// TwinCAT 3 PLC project Sys1_Inbound
// ProgramVersion: 3.1.4026.26
// libraries:
//   Tc2_Standard, * (Beckhoff Automation GmbH)
//   Tc2_System, * (Beckhoff Automation GmbH)
// project tree:
//   DUTs/ Auto_Test_DB_DUT.TcDUT (not stored), Auto_Test_DUT.TcDUT (not stored), Barcode_Station_DUT.TcDUT (not stored), Charger_DUT.TcDUT (not stored), Gate_Station_DUT.TcDUT (not stored), Level_Keys_DUT.TcDUT
//   DUTs/Conveyors/ Buffer_Cnv_Control_DUT.TcDUT (not stored), Buffer_Cnv_Inputs_DUT.TcDUT (not stored), Buffer_Cnv_Settings_DUT.TcDUT (not stored), Cnv_Errors_DUT.TcDUT (not stored), Cnv_Inputs_DUT.TcDUT (not stored), Cnv_Instruction_DUT.TcDUT (not stored), Cnv_Level_Control_DUT.TcDUT (not stored), Cnv_Level_Inputs_DUT.TcDUT, Cnv_Level_Settings_DUT.TcDUT (not stored), Cnv_Motor_DUT.TcDUT (not stored), Cnv_VTD_Control_DUT.TcDUT (not stored), Cnv_VTD_Settings_DUT.TcDUT (not stored), ECnv_Control_DUT.TcDUT (not stored), ECnv_Settings_DUT.TcDUT
//   DUTs/Safety_Stops/ Sfts_Control_DUT.TcDUT, Sfts_Inputs_DUT.TcDUT, Sfts_Instruction_DUT.TcDUT (not stored), Sfts_Settings_DUT.TcDUT (not stored)
//   DUTs/System/ ID_Decoded_DUT.TcDUT (not stored), OrderTable_DUT.TcDUT (not stored), System_DUT.TcDUT (not stored), System_Settings_DUT.TcDUT (not stored), WMS_OPC_UA_DUT.TcDUT (not stored)
//   DUTs/VTD/ VTD_Control_DUT.TcDUT (not stored), VTD_Errors_DUT.TcDUT, VTD_Inputs_DUT.TcDUT (not stored), VTD_Instruction_DUT.TcDUT, VTD_Levels_DUT.TcDUT (not stored), VTD_Motor_DUT.TcDUT, VTD_Outputs_DUT.TcDUT (not stored), VTD_Settings_DUT.TcDUT (not stored), VTD_Shuttle_Interlock_DUT.TcDUT (not stored)
//   GVLs/ Bypass.TcGVL (not stored), CNV_HMI_IO.TcGVL (not stored), Control.TcGVL (not stored), Errors.TcGVL (not stored), Force.TcGVL (not stored), Settings.TcGVL (not stored), System_Control.TcGVL (not stored)
//   GVLs/HMI/ CNV_HMI.TcGVL (not stored)
//   GVLs/IO/ IO_Panel.TcGVL, IO_VFDs.TcGVL
//   / PlcTask.TcTTO (not stored)
//   POUs/Conveyors/ Buffer_Conveyor_FB.TcPOU
//   POUs/ MAIN.TcPOU (not stored), Stack_Lights_FB.TcPOU
//   POUs/System/ Conveyors_Transfer.TcPOU
//   POUs/System/Functions/ ID_Decode_F.TcPOU (not stored), Set_Bit_F.TcPOU
//   POUs/VTD/ Light_Bars_FB.TcPOU, VTD_FB.TcPOU
// real-time tasks:
//   TASK PlcTask: cycle T#10ms, priority 20, ADS port 350
//   TASK PlcTask1: cycle T#10ms, priority 21, ADS port 351
// I/O:
//   DEVICE VTD_1 (EtherCAT), AmsNetId 192.168.0.103.2.1
//     DI-01 (EPP1008-0022) [EPP1008-0022 8 Ch. Dig. Input 24V, 3ms, M12]
//     DI-02 (EPP1008-0022) [EPP1008-0022 8 Ch. Dig. Input 24V, 3ms, M12]
//     DI-03 (EPP1008-0022) [EPP1008-0022 8 Ch. Dig. Input 24V, 3ms, M12]
//     DI-04 (EPP1008-0022) [EPP1008-0022 8 Ch. Dig. Input 24V, 3ms, M12]
//     DI-05 (EPP1008-0022) [EPP1008-0022 8 Ch. Dig. Input 24V, 3ms, M12]
//     DI-06 (EPP1008-0022) [EPP1008-0022 8 Ch. Dig. Input 24V, 3ms, M12]
//     DI-07 (EPP1008-0022) [EPP1008-0022 8 Ch. Dig. Input 24V, 3ms, M12]
//     DI-08 (EPP1008-0022) [EPP1008-0022 8 Ch. Dig. Input 24V, 3ms, M12]
//     DI-09 (EPP1008-0022) [EPP1008-0022 8 Ch. Dig. Input 24V, 3ms, M12]
//     DI-10 (EPP1008-0022) [EPP1008-0022 8 Ch. Dig. Input 24V, 3ms, M12]
//     ENCODER (EPP5001-0002) [EPP5001-0002 1Ch. SSI Encoder]
//     DIO-01 (EPP2328-0002) [EPP2328-0002 4 CH. Dig. In, 3ms, 4 Ch. Dig. Out 24V, 2A, M12]
//     DIO-02 (EPP2328-0002) [EPP2328-0002 4 CH. Dig. In, 3ms, 4 Ch. Dig. Out 24V, 2A, M12]
//     DIO-03 (EPP2328-0002) [EPP2328-0002 4 CH. Dig. In, 3ms, 4 Ch. Dig. Out 24V, 2A, M12]
//     DIO-04 (EPP2328-0002) [EPP2328-0002 4 CH. Dig. In, 3ms, 4 Ch. Dig. Out 24V, 2A, M12]
//     DIO-05 (EPP2328-0002) [EPP2328-0002 4 CH. Dig. In, 3ms, 4 Ch. Dig. Out 24V, 2A, M12]
//     DIO-06 (EPP2328-0002) [EPP2328-0002 4 CH. Dig. In, 3ms, 4 Ch. Dig. Out 24V, 2A, M12]
//     DIO-07 (EPP2328-0002) [EPP2328-0002 4 CH. Dig. In, 3ms, 4 Ch. Dig. Out 24V, 2A, M12]
//     DI-11 (EPP1809-0022) [EPP1809-0022 16 Ch. Dig. Input 24V, 3ms, M8]
//     FDI-01 (EP1918-0002) [EP1918, 8Ch. Safety Input 24V, TwinSAFE]
//       modules: Module 1 (FSOE), Module 2 (FSLOGIC)
//     PLC_IOs (EK1200) [EK1200-5000 EtherCAT Power supply (2A E-Bus)]
//       DI-01 (EL1809) [EL1809 16Ch. Dig. Input 24V, 3ms]
//       DI-02 (EL1809) [EL1809 16Ch. Dig. Input 24V, 3ms]
//       DO-01 (EL2809) [EL2809 16Ch. Dig. Output 24V, 0.5A]
//       DO-02 (EL2809) [EL2809 16Ch. Dig. Output 24V, 0.5A]
//       F-PLC (EL6910) [EL6910, TwinSAFE PLC]
//       FDI-01 (EL1918) [EL1918, 8Ch. Safety Input 24V, TwinSAFE]
//         modules: Module 1 (FSOE), Module 2 (FSLOGIC)
//       FDO-01 (EL2912) [EL2912, 2Ch. Safety Output 24V, 2A, TwinSAFE]
//         modules: Module 1 (FSOE), Module 2 (FSOUT), Module 3 (DEVICEIO), Module 4 (FSLOGIC)
//       ETHERCAT-1 (EK1322) [EK1322 2-port EtherCAT P junction with feed-in]
//       ETHERCAT-2 (EK1322) [EK1322 2-port EtherCAT P junction with feed-in]
//       ETHERCAT-3 (EK1322) [EK1322 2-port EtherCAT P junction with feed-in]
//       PROFNET (EL6633) [EL6633 PROFINET IO Controller]
//       ETHERCAT-4 (EK1122) [EK1122 2 port EtherCAT junction]
//       POWER_SUPPLY (EL9410) [EL9410 E-Bus Power Supplier  (Diagnostics)]
//       END_TERMINAL (EL9011) [EL9011 End Terminal]
//   DEVICE MAIN (EtherCAT), AmsNetId 192.168.0.103.3.1
//     PLC_IOs (EK1200) [EK1200-5000 EtherCAT Power supply (2A E-Bus)]
//       DI-01 (EL1809) [EL1809 16Ch. Dig. Input 24V, 3ms]
//       DI-02 (EL1809) [EL1809 16Ch. Dig. Input 24V, 3ms]
//       DO-01 (EL2809) [EL2809 16Ch. Dig. Output 24V, 0.5A]
//       DO-02 (EL2809) [EL2809 16Ch. Dig. Output 24V, 0.5A]
//       F-PLC (EL6910) [EL6910, TwinSAFE PLC]
//       FDI-01 (EL1918) [EL1918, 8Ch. Safety Input 24V, TwinSAFE]
//         modules: Module 1 (FSOE), Module 2 (FSLOGIC)
//       FDI-02 (EL1918) [EL1918, 8Ch. Safety Input 24V, TwinSAFE]
//         modules: Module 1 (FSOE), Module 2 (FSLOGIC)
//       FDO-01 (EL2912) [EL2912, 2Ch. Safety Output 24V, 2A, TwinSAFE]
//         modules: Module 1 (FSOE), Module 2 (FSOUT), Module 3 (DEVICEIO), Module 4 (FSLOGIC)
//       FDO-02 (EL2912) [EL2912, 2Ch. Safety Output 24V, 2A, TwinSAFE]
//         modules: Module 1 (FSOE), Module 2 (FSOUT), Module 3 (DEVICEIO), Module 4 (FSLOGIC)
//       POWER_SUPPLY (EL9410) [EL9410 E-Bus Power Supplier  (Diagnostics)]
//       PROFNET (EL6633) [EL6633 PROFINET IO Controller]
//       ETHERCAT (EK1322) [EK1322 2-port EtherCAT P junction with feed-in]
//       END_TERMINAL (EL9011) [EL9011 End Terminal]

// ---- DUTs/Conveyors/Cnv_Level_Inputs_DUT.TcDUT
TYPE Cnv_Level_Inputs_DUT :
STRUCT
	Cnv1_Inputs:	Buffer_Cnv_Inputs_DUT;
	Cnv2_Inputs:	Buffer_Cnv_Inputs_DUT;
END_STRUCT
END_TYPE

// ---- DUTs/Conveyors/ECnv_Settings_DUT.TcDUT
TYPE ECnv_Settings_DUT :
STRUCT
	ID:	DINT;
	Barcode_ID:	UINT;
	Cnv_Level:	UINT;
	TC_Time:	UINT;
	Transfer_Time:	UINT;
	Pallet_Align_Time:	UINT;
	Slow_Speed:	UINT;
	Full_Speed:	UINT;
	Manual_Speed:	UINT;
END_STRUCT
END_TYPE

// ---- DUTs/Level_Keys_DUT.TcDUT
TYPE Level_Keys_DUT :
STRUCT
	Level:	ARRAY[1..6] OF BOOL;
END_STRUCT
END_TYPE

// ---- DUTs/Safety_Stops/Sfts_Control_DUT.TcDUT
TYPE Sfts_Control_DUT :
STRUCT
	Mode:  UINT;
	Error:  BOOL;
	Enabled:  Bool;
	Running:  Bool;
	LP_State:  USInt;
	Motor_Extend:  Bool;
	Motor_Retract:  Bool;
	SM_State:  UInt;
	Instruction:  Sfts_Instruction_DUT;
	Inputs:  Sfts_Inputs_DUT;
END_STRUCT
END_TYPE

// ---- DUTs/Safety_Stops/Sfts_Inputs_DUT.TcDUT
TYPE Sfts_Inputs_DUT :
STRUCT
	DP_Extended:  BOOL;
	DP_Retracted:  Bool;
END_STRUCT
END_TYPE

// ---- DUTs/VTD/VTD_Errors_DUT.TcDUT
TYPE VTD_Errors_DUT :
STRUCT
	Error_Word_1:	UINT;
	Error_Word_2:	UINT;
	Error_Word_3:	UINT;
	Error_Word_4:	UINT;
	Error_Word_5:	UINT;
END_STRUCT
END_TYPE

// ---- DUTs/VTD/VTD_Instruction_DUT.TcDUT
TYPE VTD_Instruction_DUT :
STRUCT
	Mode_Change:  UINT;
	Stop:  BOOL;
	Enable:  Bool;
	Execulte:  Bool;
	Reset:  Bool;
	Pallet_Type:  UInt;
	Task_ID:  UInt;
	Task_Metadata:  String;
	Move_To_Level:  UInt;
	Manual_Up:  Bool;
	Manual_Down:  Bool;
	Manual_LP_Retract:  Bool;
	Manual_LP_Extend:  Bool;
	Start_Teach:  BOOL;
END_STRUCT
END_TYPE

// ---- DUTs/VTD/VTD_Motor_DUT.TcDUT
TYPE VTD_Motor_DUT :
STRUCT
	Enable:  BOOL;
	Enabled:  BOOL;
	Ready:  Bool;
	Running:  Bool;
	Forward:  Bool;
	Reverse:  Bool;
	Brake_Opened:  Bool;
	Speed:  Int;
	Speed_Actual:  Int;
	Actual_Current:  Int;
	Actual_Torque:  UInt;
	Acc_Factor:  UInt;
	Config_Axis:  Word;
	Error:  Bool;
	Status:  Word;
	Communication_Error:  Word;
	Lockout:  BOOL;
END_STRUCT
END_TYPE

// ---- GVLs/IO/IO_Panel.TcGVL
{attribute 'qualified_only'}
VAR_GLOBAL
	C1112_VTD_CIRCUIT_BREAKER AT%I*:BOOL;
	

END_VAR

// ---- GVLs/IO/IO_VFDs.TcGVL
{attribute 'qualified_only'}
VAR_GLOBAL
	
END_VAR

// ---- POUs/Conveyors/Buffer_Conveyor_FB.TcPOU
FUNCTION_BLOCK Buffer_Conveyor_FB
VAR_INPUT
	Cnv_Settings:  Buffer_Cnv_Settings_DUT;
	VTD_Level:  UINT;
	Safety_OK:  Bool;
	CNV_In_Out:  Bool;
	CNV1_2_Selected:  UInt;
	Time_CheckPallet:  Time;
	Time_CheckNoPallet:  TIME;
END_VAR
VAR_OUTPUT
END_VAR
VAR_IN_OUT
	Cnv_Control:  Buffer_Cnv_Control_DUT;
END_VAR
VAR
	State:  UINT;
	Timer_Transfer:  TON;
	Watchdog:  TON;
	Transfer_Direction:  String;
	MainSetpoint:  Int;
	R_Automatic_Mode:  R_TRIG;
	R_Start_DB:  R_TRIG;
	R_Stop_DB:  R_TRIG;
	ID_Decoded:  ID_Decoded_DUT;
	ID_Decoded_From:  ID_Decoded_DUT;
	ID_Decoded_To:  ID_Decoded_DUT;
	T_Ramp:  TON;
	HMI_Reset:  Bool;
	T_CheckNoPallet:  TON;
	Time_SlowDown_Ramp:  Time;
	T_CheckPallet:  TON;
END_VAR
VAR_TEMP
	Execute_Old:  BOOL;
	Stop_Old:  BOOL;
	Forward:  Bool;
	Backward:  Bool;
	SftyPinUp:  Bool;
	SftyPinDown:  BOOL;
END_VAR

R_Start_DB(CLK := Cnv_Control.Instruction.Execute AND NOT Execute_Old);
R_Stop_DB(CLK := Cnv_Control.Instruction.Stop AND NOT Stop_Old);

Execute_Old := Cnv_Control.Instruction.Execute;
Stop_Old := Cnv_Control.Instruction.Stop;

Cnv_Control.Enabled := Cnv_Control.Instruction.Enable OR Cnv_Control.Mode = 3;

ID_Decode_F(ID := Cnv_Settings.ID,
            ID_Decoded := ID_Decoded);

ID_Decode_F(ID := Cnv_Control.Instruction.Transfer_From_ID,
              ID_Decoded := ID_Decoded_From);

ID_Decode_F(ID := Cnv_Control.Instruction.Transfer_To_ID,
              ID_Decoded := ID_Decoded_To);

//MODES
Cnv_Control.Mode := Cnv_Control.Instruction.Mode_Change;
IF (Cnv_Control.Mode = 1 OR Cnv_Control.Mode = 5) AND NOT Cnv_Control.Error THEN
    State := 500;
END_IF;

R_Automatic_Mode(CLK := Cnv_Control.Mode = 3);
IF R_Automatic_Mode.Q OR (NOT Cnv_Control.Enabled AND NOT Cnv_Control.Error) THEN
    State := 0;
END_IF;

(*
Mode select is done via the HMI. Might add external mode select switches.
        
        Mode select mask:
        0: Disabled
        1: Manual
        2: Semi-Auto
        3: Auto
        4: Teach - N/A for Cnv
        5: Maintenance
        
Device ID Format: XXYYZZ    
XX = Device type   
    40  VTD
    10  Cnv_Front_of_VTD
    11  Cnv_Rear_of_VTD
    12  Cnv_On_Extractor
    20  Safety_Stop_Front_of_VTD
    21  Safety_Stop_Rear_of_VTD
  
YY = Floor   
ZZ = VTD Connected to    
Example: 110203 Conveyor at the rear of VTD 3 on level 2    
*)

{REGION Sensor allocations}
    //PALLET DETECT
    Forward := Cnv_Control.Inputs.Forward_Sensor;
    Backward := Cnv_Control.Inputs.Backward_Sensor;
    
    //SAFETY PINS (IT DOESN'T EXIST IN ECONVEYORS)
    SftyPinUp := Cnv_Control.Safety_Stop_Cnrl.Inputs.DP_Extended;
    SftyPinDown := Cnv_Control.Safety_Stop_Cnrl.Inputs.DP_Retracted;
{END_REGION}

{REGION Cyclic Checks} 
    // Check Pallet
    T_CheckPallet(IN:=Forward AND Backward,
                   PT:=Time_CheckPallet);
    
    T_CheckNoPallet(IN:=Cnv_Control.Running AND NOT Forward AND NOT Backward,
                   PT:=Time_CheckNoPallet);
    
    //Conditions for Conveyor occupied
  IF T_CheckPallet.Q OR // Both sensors triggered after a timer
        (NOT Forward AND Backward AND NOT Cnv_Control.Running) OR //Forward sensor triggered and not running
        (Forward AND NOT Backward AND NOT Cnv_Control.Running) //Backward sensor triggered and not running
    THEN
        Cnv_Control.Cnv_Occupied := TRUE;//Conveyor occupied
    ELSIF T_CheckNoPallet.Q OR //Check pallet Timer
        (NOT Cnv_Control.Running AND NOT Forward AND NOT Backward) //No sensor detected and Conveyor not running
    THEN
        //No Pallet
        Cnv_Control.Cnv_Occupied := FALSE;
    END_IF;
    
    // Update the Cnv_Control opbject
    Cnv_Control.SM_State := State;
    Cnv_Control.Stopped := NOT Cnv_Control.Running;
    IF Cnv_Control.Instruction.Inbound_Ready OR Cnv_Control.Instruction.Outbound_Ready THEN
        Cnv_Control.Ready_For_Task := TRUE;
    ELSE
        Cnv_Control.Ready_For_Task := FALSE;
    END_IF;
    
    IF ID_Decoded.Device_Type = 10 THEN
        Settings.LCnv_Sys[ID_Decoded.VTD].Cnv_Level[ID_Decoded.Level].Cnv1.Cnv_Level := INT_TO_UINT(ID_Decoded.Level);
    ELSIF ID_Decoded.Device_Type = 11 THEN
        Settings.LCnv_Sys[ID_Decoded.VTD].Cnv_Level[ID_Decoded.Level].Cnv2.Cnv_Level := INT_TO_UINT(ID_Decoded.Level);
    END_IF;
{END_REGION}

{REGION Auto/Semi auto mode}
    CASE State OF
        0: //Initialization
            Cnv_Control.Instruction.Inbound_Ready := FALSE;
            Cnv_Control.Instruction.Outbound_Ready := FALSE;
            Cnv_Control.Instruction.Transfer_Complete := 0;
            Cnv_Control.Instruction.Transfer_in_Progress := FALSE;
            Cnv_Control.Running := FALSE;
            Cnv_Control.Motor.Forward := FALSE;
            Cnv_Control.Motor.Reverse := FALSE;
            Cnv_Control.Motor.Speed := 0;
            Timer_Transfer(IN := FALSE,
                            PT := T#0S);
            T_Ramp(IN := FALSE,
                    PT := t#0s);
            IF Cnv_Control.Enabled AND (Cnv_Control.Mode = 3 OR Cnv_Control.Mode = 2) AND Cnv_Control.Error = 0 THEN
                State := 10;
            END_IF;
            
        10: //Standby - Conveyor ready to receive instruction
            IF Cnv_Control.Ready_For_Task AND (R_Start_DB.Q OR Cnv_Control.Instruction.Start_Transfer)
            THEN //WCS NORMAL TRANSFER
                Cnv_Control.Instruction.Inbound_Ready := FALSE;
                Cnv_Control.Instruction.Outbound_Ready := FALSE;
                Cnv_Control.Done := FALSE;
                Cnv_Control.Running := TRUE;
                Cnv_Control.Instruction.Transfer_in_Progress := TRUE;
                Cnv_Control.Current_Task_ID := Cnv_Control.Instruction.Task_ID;
                State := 20;
            ELSIF Cnv_Control.Instruction.Start_Transfer AND ID_Decoded.Level = 10 AND VTD_Level <> Cnv_Settings.Cnv_Level THEN
                //Extractor not at the correct level
                Set_Bit_F(BIT_Number := 2,
                            Variavel := Cnv_Control.Cnv_Errors.Error_Word_3);
            END_IF;
            
            //----------------------- Pallet Movement -----------------------
        20: //Set the direction of transfer
            IF ID_Decoded.Device_Type = 10 AND ID_Decoded_From.Device_Type = 12 AND NOT Cnv_Control.Cnv_Occupied AND
                Control.ECnv_Sys[ID_Decoded.VTD].Cnv_Occupied THEN //Extractor to CNV 1
                Cnv_Control.Motor.Speed := Cnv_Settings.Full_Speed;
                Cnv_Control.Motor.Forward := TRUE;
                Transfer_Direction := 'Forward';
                State := 30;
            ELSIF ID_Decoded.Device_Type = 10 AND ID_Decoded_To.Device_Type = 11 AND Cnv_Control.Cnv_Occupied AND
                NOT Control.LCnv_Sys[ID_Decoded.VTD].Cnv_Level[ID_Decoded.Level].Cnv2.Cnv_Occupied THEN // CNV 1 to CNV 2
                IF Control.LCnv_Sys[ID_Decoded.VTD].Cnv_Level[ID_Decoded.Level].Cnv2.SM_State = 30 THEN //Wait CNV 2 Run
                    Cnv_Control.Motor.Speed := Cnv_Settings.Full_Speed;
                    Cnv_Control.Motor.Forward := TRUE;
                    Transfer_Direction := 'Forward';
                    State := 30;
                END_IF;
            ELSIF ID_Decoded.Device_Type = 11 AND ID_Decoded_To.Device_Type = 10 AND Cnv_Control.Cnv_Occupied AND
                NOT Control.LCnv_Sys[ID_Decoded.VTD].Cnv_Level[ID_Decoded.Level].Cnv1.Cnv_Occupied THEN //CNV 2 To Cnv 1
                IF Control.LCnv_Sys[ID_Decoded.VTD].Cnv_Level[ID_Decoded.Level].Cnv1.SM_State = 30 THEN //Wait CNV1 RUn
                    Cnv_Control.Motor.Speed := Cnv_Settings.Full_Speed;
                    Cnv_Control.Motor.Reverse := TRUE;
                    Transfer_Direction := 'Backward';
                    State := 30;
                END_IF;
            ELSIF ID_Decoded.Device_Type = 10 AND ID_Decoded_To.Device_Type = 12 AND Cnv_Control.Cnv_Occupied AND
                NOT Control.ECnv_Sys[ID_Decoded.VTD].Cnv_Occupied THEN //CNV 1 To extractor
                IF Control.ECnv_Sys[ID_Decoded.VTD].SM_State = 30 THEN //Wait CVTD RUn
                    Cnv_Control.Motor.Speed := Cnv_Settings.Full_Speed;
                    Cnv_Control.Motor.Reverse := TRUE;
                    Transfer_Direction := 'Backward';
                    State := 30;
                END_IF;
            ELSE //14:3 Cnv cannot transfer to that location
                Set_Bit_F(BIT_Number := 5,
                            Variavel := Cnv_Control.Cnv_Errors.Error_Word_2);
            END_IF;
            
        30: // Running
            IF R_Stop_DB.Q THEN
                Cnv_Control.Motor.Forward := FALSE;
                Cnv_Control.Motor.Reverse := FALSE;
                Cnv_Control.Motor.Speed := 0;
                State := 0;
            ELSE
                //Slowdown ramp
                T_Ramp(IN := TRUE,
                        PT := Time_SlowDown_Ramp);
                IF T_Ramp.ET > (Time_SlowDown_Ramp * 70) / 100 AND T_Ramp.ET < (Time_SlowDown_Ramp * 80) / 100 THEN
                    Cnv_Control.Motor.Speed := Cnv_Settings.Slow_Speed * 3;
                ELSIF T_Ramp.ET > (Time_SlowDown_Ramp * 80) / 100 AND T_Ramp.ET < (Time_SlowDown_Ramp * 90) / 100 THEN
                    Cnv_Control.Motor.Speed := Cnv_Settings.Slow_Speed * 2;
                ELSIF T_Ramp.ET >= Time_SlowDown_Ramp THEN
                    Cnv_Control.Motor.Speed := Cnv_Settings.Slow_Speed;
                END_IF;
            END_IF;
            
            //Check conditions to stop the motor
            IF (ID_Decoded.Device_Type = 10 AND ID_Decoded_From.Device_Type = 12) OR //ECONV To CNV 1 - 10(CNV1)
                (ID_Decoded.Device_Type = 11 AND ID_Decoded_From.Device_Type = 10) OR //CNV 1 To CNV 2 - 11(CNV2)
                (ID_Decoded.Device_Type = 10 AND ID_Decoded_From.Device_Type = 11) //CNV 2 To CNV 1 - 10(CNV1)
            THEN
                IF Cnv_Control.Cnv_Occupied THEN //Stop the motor if the conveyor is not occupied anymore
                    State := 35;
                END_IF;
            ELSIF (ID_Decoded.Device_Type = 10 AND ID_Decoded_To.Device_Type = 12) OR //CNV 1 To ECNV - 10(CNV1)
                (ID_Decoded.Device_Type = 10 AND ID_Decoded_To.Device_Type = 11) OR //CNV 1 To CNV 2 - 10(CNV1)
                (ID_Decoded.Device_Type = 11 AND ID_Decoded_To.Device_Type = 10) //CNV 2 To CNV 1 - 11(CNV2)
            THEN
                IF NOT Cnv_Control.Cnv_Occupied THEN //Stop the motor if the conveyor is occupied
                    State := 35;
                END_IF;
            END_IF;
            
            //Monitor the transfer progress
            Timer_Transfer(IN := TRUE,
                            PT := UINT_TO_TIME(Cnv_Settings.Transfer_Time) * 1000);
            //If the watchdog bites, kill the process
            IF Timer_Transfer.Q THEN //14:1 Transfer timed out
                Set_Bit_F(BIT_Number := 3,
                           Variavel := Cnv_Control.Cnv_Errors.Error_Word_2);
            END_IF;
            
        35: //Stop motor
                T_Ramp(IN := FALSE,
                        PT := T#0S);
                Cnv_Control.Motor.Forward := FALSE;
                Cnv_Control.Motor.Reverse := FALSE;
                Cnv_Control.Motor.Speed := 0;
                Cnv_Control.Done := TRUE;
                State := 0;
            
        //----------------------- Pallet Alignment -----------------------
        400: //Error state
            Cnv_Control.Instruction.Inbound_Ready := FALSE;
            Cnv_Control.Instruction.Outbound_Ready := FALSE;
            Cnv_Control.Running := FALSE;
            Cnv_Control.Motor.Speed := 0;
            Cnv_Control.Motor.Forward := FALSE;
            Cnv_Control.Motor.Reverse := FALSE;
            Cnv_Control.Instruction.Stop := FALSE;
            Cnv_Control.Instruction.Transfer_in_Progress := FALSE;
            Watchdog(IN := FALSE,
                      PT := T#0S);
            Timer_Transfer(IN := FALSE,
                            PT := T#0S);

            T_Ramp(IN := FALSE,
                    PT := t#0s);
            IF Cnv_Control.Instruction.Reset OR SYSTEM_CONTROL.Reset_All OR HMI_Reset THEN
                Cnv_Control.Warning := 0;
                Cnv_Control.Current_Task_ID := 0;
                Cnv_Control.Error := FALSE; //Reset the conveyor
                
                Cnv_Control.Cnv_Errors.Error_Word_1 := 0;
                Cnv_Control.Cnv_Errors.Error_Word_2 := 0;
                Cnv_Control.Cnv_Errors.Error_Word_3 := 0;
                Cnv_Control.Cnv_Errors.Error_Word_4 := 0;
                State := 0;
            END_IF;
            
        500:
            IF Cnv_Control.Enabled THEN
                IF Cnv_Control.Instruction.Foward OR
                    (ID_Decoded.Device_Type = 10 AND Cnv_Control.Instruction.Start_Transfer AND NOT CNV_In_Out AND CNV1_2_Selected = 1 (*RECEIVE = 0*)) OR
                    (ID_Decoded.Device_Type = 10 AND Cnv_Control.Instruction.Start_Transfer AND CNV_In_Out AND CNV1_2_Selected = 2 (*SEND = 1*)) OR
                    (ID_Decoded.Device_Type = 11 AND Cnv_Control.Instruction.Start_Transfer AND NOT CNV_In_Out AND NOT Forward (*RECEIVE = 0*))
                THEN
                    Cnv_Control.Motor.Speed := Cnv_Settings.Manual_Speed;
                    Cnv_Control.Motor.Forward := TRUE;
                    Cnv_Control.Running := TRUE;
                ELSIF Cnv_Control.Instruction.Backward OR
                    (ID_Decoded.Device_Type = 10 AND Cnv_Control.Instruction.Start_Transfer AND NOT CNV_In_Out AND CNV1_2_Selected = 2 (*RECEIVE = 0*)) OR
                    (ID_Decoded.Device_Type = 10 AND Cnv_Control.Instruction.Start_Transfer AND CNV_In_Out AND CNV1_2_Selected = 1 (*SEND = 1*)) OR
                    (ID_Decoded.Device_Type = 11 AND Cnv_Control.Instruction.Start_Transfer AND CNV_In_Out (*SEND = 1*))
                THEN
                    Cnv_Control.Motor.Speed := Cnv_Settings.Manual_Speed;
                    Cnv_Control.Motor.Reverse := TRUE;
                    Cnv_Control.Running := TRUE;
                ELSE
                    Cnv_Control.Motor.Speed := 0;
                    Cnv_Control.Motor.Forward := FALSE;
                    Cnv_Control.Motor.Reverse := FALSE;
                    Cnv_Control.Running := FALSE;
                END_IF;
            END_IF;
            IF Cnv_Control.Mode <> 1 AND Cnv_Control.Mode <> 5 THEN
                State := 0;
            END_IF;
    END_CASE;
{END_REGION}

{REGION Cyclic Error Checks}
    IF NOT Safety_OK THEN //11:1
        Set_Bit_F(BIT_Number := 0,
                    Variavel := Cnv_Control.Cnv_Errors.Error_Word_1);
    END_IF;
    
    IF Cnv_Control.Motor.Error THEN
        Set_Bit_F(BIT_Number:= 0,
                  Variavel := Cnv_Control.Cnv_Errors.Error_Word_4);
    END_IF;
    
    IF Cnv_Control.Instruction.Stop THEN //HMI STOP
        Set_Bit_F(BIT_Number := 1,
                    Variavel := Cnv_Control.Cnv_Errors.Error_Word_1);
    END_IF;
    
    IF Cnv_Control.Safety_Stop_Cnrl.Error THEN
        Set_Bit_F(BIT_Number := 1,
                    Variavel := Cnv_Control.Cnv_Errors.Error_Word_4);
    END_IF;
    
    IF ((ID_Decoded.VTD = 1 AND ERRORS.Errors_Profinet_1.8) OR
        (ID_Decoded.VTD = 2 AND Errors_Profinet_3.7)) AND Cnv_Control.Mode <> 1
    THEN //Profinet error
        Set_Bit_F(BIT_Number := 3,
                    Variavel := Cnv_Control.Cnv_Errors.Error_Word_3);
    END_IF;
    
    
    // go to error state
    IF Cnv_Control.Cnv_Errors.Error_Word_1 <> 0 OR
        Cnv_Control.Cnv_Errors.Error_Word_2 <> 0 OR
        Cnv_Control.Cnv_Errors.Error_Word_3 <> 0 OR
        Cnv_Control.Cnv_Errors.Error_Word_4 <> 0
    THEN
        Cnv_Control.Error := TRUE;
        State := 400;
    END_IF;
{END_REGION}

{REGION VFD}
    //Status
    Cnv_Control.Motor.Ready := (Cnv_Control.Inputs.VFD_Status.%X0 OR Cnv_Control.Inputs.VFD_Status.%X1) AND NOT Cnv_Control.Motor.Error;
    Cnv_Control.Motor.Error := Cnv_Control.Inputs.VFD_Status.%X3 OR Cnv_Control.Inputs.VFD_Status.%X7 OR NOT Cnv_Control.Inputs.VFD_Status.%X13;
    Cnv_Control.Motor.Enabled := Cnv_Control.Inputs.VFD_Status.%X2;
    Cnv_Control.Motor.Actual_Current := SCALE_X(MIN := 0,
                                                 VALUE := NORM_X(MIN := 0,
                                                                 VALUE := Cnv_Control.Inputs.VFD_ActualCurrent,
                                                                 MAX := 16384),
                                                 MAX := 1.98);
    
    
    //Actual Speed
    IF MainSetpoint > 0 THEN
        Cnv_Control.Motor.Speed_Actual := SCALE_X(MIN := 0,
                                                   VALUE := NORM_X(MIN := 0,
                                                                   VALUE := Cnv_Control.Inputs.VFD_Speed_Actual,
                                                                   MAX := 16384),
                                                   MAX := 130);
        
        Cnv_Control.Motor.Actual_Torque := SCALE_X(MIN := 0,
                                                    VALUE := NORM_X(MIN := 0,
                                                                    VALUE := Cnv_Control.Inputs.VFD_ActualTorque,
                                                                    MAX := 16384),
                                                    MAX := 100);
    ELSIF MainSetpoint < 0 THEN
        Cnv_Control.Motor.Speed_Actual := SCALE_X(MIN := 0,
                                                   VALUE := NORM_X(MIN := 0,
                                                                   VALUE := Cnv_Control.Inputs.VFD_Speed_Actual * -1,
                                                                   MAX := 16384),
                                                   MAX := 130);
        
        Cnv_Control.Motor.Actual_Torque := SCALE_X(MIN := 0,
                                                    VALUE := NORM_X(MIN := 0,
                                                                    VALUE := Cnv_Control.Inputs.VFD_ActualTorque * -1,
                                                                    MAX := 16384),
                                                    MAX := 100);
    ELSE
        Cnv_Control.Motor.Speed_Actual := 0;
        Cnv_Control.Motor.Actual_Torque := 0;
    END_IF;
    
    //MAIN SETPOINT
    IF Cnv_Control.Motor.Forward THEN
        MainSetpoint := (SCALE_X(MIN := 0,
                                  VALUE := NORM_X(MIN := 0,
                                                  VALUE := Cnv_Control.Motor.Speed (** 1.681*),
                                                  MAX := 130),
                                  MAX := 1865.0) * -1);
    ELSIF Cnv_Control.Motor.Reverse THEN
        MainSetpoint := SCALE_X(MIN := 0,
                                 VALUE := NORM_X(MIN := 0,
                                                 VALUE := Cnv_Control.Motor.Speed (** 1.681*),
                                                 MAX := 130),
                                 MAX := 1865.0);
    ELSE
        MainSetpoint := 0;
    END_IF;
    
    SinaSpeed(EnableAxis := Cnv_Control.Motor.Forward OR Cnv_Control.Motor.Reverse,
               AckError := Cnv_Control.Instruction.Reset OR "Reset_All" OR HMI_Reset,
               SpeedSp := MainSetpoint,
               RefSpeed := 1865.0,
               HWIDSTW := Cnv_Settings.G120_Hardware_ID,
               HWIDZSW := Cnv_Settings.G120_Hardware_ID);
{END_REGION}

HMI_Reset := "Screen_DB_1".Reset_All[1] OR "Screen_DB_1".Reset_All[2] OR "CNV_HMI"."Reset(1)"[1] OR "CNV_HMI"."Reset(1)"[2];
;

END_FUNCTION_BLOCK

// ---- POUs/System/Functions/Set_Bit_F.TcPOU
FUNCTION Set_Bit_F : BOOL
VAR_INPUT
	BIT_Number:  UINT;
END_VAR
VAR
END_VAR
VAR_IN_OUT
	Variavel: WORD;
END_VAR

// Set the bit
Variavel := Variavel OR SHL(WORD#1,BIT_Number);

END_FUNCTION

// ---- POUs/Stack_Lights_FB.TcPOU
FUNCTION_BLOCK Stack_Lights_FB
VAR_INPUT
	System_Auto:  BOOL;
	Fault:  BOOL;
END_VAR
VAR_OUTPUT
	Red:  BOOL;
	Green:  BOOL;
	Orange:  BOOL;
END_VAR
VAR
END_VAR

//Commands for Stack Light

IF Fault THEN  // Fault = Red
    Red := "Clock_0.5Hz";
    Green := FALSE;
    Orange := FALSE;
ELSIF System_Auto THEN  // (1)Manual = Yellow
    Orange := FALSE;
    Red := FALSE;
    Green := TRUE;
ELSIF NOT System_Auto THEN  // (2)Semi-Auto = Blue
    Green := FALSE;
    Orange := TRUE;
    Red := FALSE;
// ELSIF System_Auto = 3 THEN  // (3)Auto = Green
//     Green := FALSE;
//     Red := FALSE;
//     Yellow := TRUE;

ELSE
    Green := FALSE;
    Red := FALSE;
    Orange := FALSE;
END_IF;

END_FUNCTION_BLOCK

// ---- POUs/System/Conveyors_Transfer.TcPOU
FUNCTION Conveyors_Transfer : BOOL
VAR_INPUT
END_VAR
VAR
	i_Lev:  UINT;
	i_Sys:  UINT;
	Concat1:  String;
	Concat2:  String;
	ID:  DInt;
	StrLev:  String;
	StrSys:  String;
	Level:  UINT;
END_VAR

FOR i_Sys := 1 TO 2 DO
    StrSys := UINT_TO_STRING(i_Sys);
    // Remove "+"
    IF StrSys[1] = '+' THEN
        StrSys := RIGHT(StrSys, L := LEN(StrSys) - 1);
    END_IF;
    
    {region "ID OF THE VTD CONVEYOR"}
        FOR i_Lev := Settings.VTD_Sys[i_Sys].Lowest_Level TO Settings.VTD_Sys[i_Sys].Highest_Level DO
            IF (i_Sys >= 1) AND (i_Sys <= 2) THEN
                IF Control.VTD_Sys[i_Sys].Current_Level = i_Lev THEN
                    StrLev := UINT_TO_STRING(i_Lev);
                    
                    // Remove "+"
                    IF StrLev[1] = '+' THEN
                        StrLev := RIGHT(StrLev, L := LEN(StrLev) - 1);
                    END_IF;
                    
                    //Build ID
                    Concat1 := CONCAT('120', StrLev);
                    Concat2 := CONCAT(Concat1, '0');
                    ID := STRING_TO_DINT(CONCAT(Concat2, StrSys));
                    
                    Settings.ECnv_Sys[i_Sys].ID := ID;
                    Settings.ECnv_Sys[i_Sys].Cnv_Level := i_Lev;
                END_IF;
            END_IF;
        END_FOR;
    {endregion}
        
        {region "READY TO RECEIVE"}
            //EXTRACTOR CONVEYOR
            FOR i_Lev := 2 TO Settings.VTD_Sys[i_Sys].Highest_Level DO
                IF Control.VTD_Sys[i_Sys].Current_Level = i_Lev THEN
                    StrLev := UINT_TO_STRING(i_Lev);
                    
                    // Remove "+"
                    IF StrLev[1] = '+' THEN
                        StrLev := RIGHT(StrLev, L := LEN(StrLev) - 1);
                    END_IF;
                    
                    //Build ID
                    Concat1 := CONCAT('120', StrLev);
                    Concat2 := CONCAT(Concat1, '0');
                    ID := STRING_TO_DINT(CONCAT(Concat2, StrSys));
                END_IF;
                
                IF Settings.ECnv_Sys[i_Sys].ID = ID AND NOT Control.ECnv_Sys[i_Sys].Error AND NOT Control.ECnv_Sys[i_Sys].Running
                    AND NOT Control.ECnv_Sys[i_Sys].Cnv_Occupied AND NOT Control.ECnv_Sys[i_Sys].Instruction.Outbound_Ready AND
                    NOT Control.LCnv_Sys[i_Sys].Cnv_Level[i_Lev].Cnv1.Running AND
                    (Control.ECnv_Sys[i_Sys].Mode = 2 OR Control.ECnv_Sys[i_Sys].Mode = 3) THEN
                    Control.ECnv_Sys[i_Sys].Instruction.Inbound_Ready := TRUE;
                END_IF;
            END_FOR;
            
            //BUFFER CONVEYORS
            FOR i_Lev := 2 TO Settings.VTD_Sys[i_Sys].Highest_Level DO
                //CNV 1
                IF NOT Control.LCnv_Sys[i_Sys].Cnv_Level[i_Lev].Cnv1.Error AND
                    NOT Control.LCnv_Sys[i_Sys].Cnv_Level[i_Lev].Cnv1.Running AND
                    NOT Control.LCnv_Sys[i_Sys].Cnv_Level[i_Lev].Cnv1.Cnv_Occupied AND
                    NOT Control.LCnv_Sys[i_Sys].Cnv_Level[i_Lev].Cnv1.Instruction.Outbound_Ready AND
                    (Control.LCnv_Sys[i_Sys].Cnv_Level[i_Lev].Cnv1.Mode = 2 OR Control.LCnv_Sys[i_Sys].Cnv_Level[i_Lev].Cnv1.Mode = 3) AND
                    NOT Control.ECnv_Sys[i_Sys].Running AND NOT Control.LCnv_Sys[i_Sys].Cnv_Level[i_Lev].Cnv2.Running
                THEN
                    Control.LCnv_Sys[i_Sys].Cnv_Level[i_Lev].Cnv1.Instruction.Inbound_Ready := TRUE;
                END_IF;
                
                //CNV 2
                IF NOT Control.LCnv_Sys[i_Sys].Cnv_Level[i_Lev].Cnv2.Error AND
                    NOT Control.LCnv_Sys[i_Sys].Cnv_Level[i_Lev].Cnv2.Running AND
                    NOT Control.LCnv_Sys[i_Sys].Cnv_Level[i_Lev].Cnv2.Cnv_Occupied AND
                    NOT Control.LCnv_Sys[i_Sys].Cnv_Level[i_Lev].Cnv2.Instruction.Outbound_Ready AND
                    (Control.LCnv_Sys[i_Sys].Cnv_Level[i_Lev].Cnv2.Mode = 2 OR Control.LCnv_Sys[i_Sys].Cnv_Level[i_Lev].Cnv2.Mode = 3) THEN
                    Control.LCnv_Sys[i_Sys].Cnv_Level[i_Lev].Cnv2.Instruction.Inbound_Ready := TRUE;
                END_IF;
            END_FOR;
        {endregion}
        
        {region "READY TO SEND"}
            //EXTRACTOR CONVEYOR
            Level := Settings.ECnv_Sys[i_Sys].Cnv_Level;
            
            IF Settings.ECnv_Sys[i_Sys].Cnv_Level >= 2 AND
                Settings.ECnv_Sys[i_Sys].Cnv_Level <= Settings.VTD_Sys[i_Sys].Highest_Level AND //Leveled
                Control.ECnv_Sys[i_Sys].Cnv_Occupied AND //Econveyor occupied
                NOT Control.ECnv_Sys[i_Sys].Error AND //not error
                NOT Control.ECnv_Sys[i_Sys].Running AND //not RUNNING
                Control.LCnv_Sys[i_Sys].Cnv_Level[Level].Cnv1.Instruction.Inbound_Ready AND 
                (Control.LCnv_Sys[i_Sys].Cnv_Level[Level].Cnv1.Mode = 2 OR
                Control.LCnv_Sys[i_Sys].Cnv_Level[Level].Cnv1.Mode = 3)  AND //cnv1 semi or auto mode
                (Control.ECnv_Sys[i_Sys].Mode = 2 OR Control.ECnv_Sys[i_Sys].Mode = 3) THEN //Econveyor semi or auto mode 
                Control.ECnv_Sys[i_Sys].Instruction.Outbound_Ready := TRUE;
            END_IF;
            
            
            //BUFFER CONVEYORS
            FOR i_Lev := 2 TO Settings.VTD_Sys[i_Sys].Highest_Level DO
                //CNV 1
                IF ((Control.ECnv_Sys[i_Sys].Instruction.Inbound_Ready AND Control.VTD_Sys[i_Sys].Current_Level = i_Lev) OR
                    Control.LCnv_Sys[i_Sys].Cnv_Level[i_Lev].Cnv2.Instruction.Inbound_Ready) AND //Extractor or CNV 2, inbound ready
                    
                    NOT Control.LCnv_Sys[i_Sys].Cnv_Level[i_Lev].Cnv2.Instruction.Transfer_in_Progress AND //NOT CNV2 transfer in progress
                    Control.LCnv_Sys[i_Sys].Cnv_Level[i_Lev].Cnv1.Cnv_Occupied AND //Not occupied
                    NOT Control.LCnv_Sys[i_Sys].Cnv_Level[i_Lev].Cnv1.Error AND NOT Control.LCnv_Sys[i_Sys].Cnv_Level[i_Lev].Cnv1.Running AND //NOT error and NOT running
                    (Control.LCnv_Sys[i_Sys].Cnv_Level[i_Lev].Cnv1.Mode = 2 OR Control.LCnv_Sys[i_Sys].Cnv_Level[i_Lev].Cnv1.Mode = 3)//Semi auto or auto
                THEN 
                    Control.LCnv_Sys[i_Sys].Cnv_Level[i_Lev].Cnv1.Instruction.Outbound_Ready := TRUE;
                END_IF;
                
                //CNV 2
                IF Control.LCnv_Sys[i_Sys].Cnv_Level[i_Lev].Cnv1.Instruction.Inbound_Ready AND //CNV 1, inbound ready
                    NOT Control.LCnv_Sys[i_Sys].Cnv_Level[i_Lev].Cnv1.Instruction.Transfer_in_Progress AND //NOT CNV 1 transfer in progress
                    Control.LCnv_Sys[i_Sys].Cnv_Level[i_Lev].Cnv2.Cnv_Occupied AND //Not occupied
                    NOT Control.LCnv_Sys[i_Sys].Cnv_Level[i_Lev].Cnv2.Error AND NOT Control.LCnv_Sys[i_Sys].Cnv_Level[i_Lev].Cnv2.Running AND //NOT error and NOT running
                    (Control.LCnv_Sys[i_Sys].Cnv_Level[i_Lev].Cnv2.Mode = 2 OR Control.LCnv_Sys[i_Sys].Cnv_Level[i_Lev].Cnv2.Mode = 3)//Semi auto or auto
                THEN
                    Control.LCnv_Sys[i_Sys].Cnv_Level[i_Lev].Cnv2.Instruction.Outbound_Ready := TRUE;
                END_IF;
            END_FOR;
       {endregion}
    END_FOR;

END_FUNCTION

// ---- POUs/VTD/Light_Bars_FB.TcPOU
FUNCTION_BLOCK Light_Bars_FB
VAR_INPUT
	VTD_Mode:  UINT;
	VTD_Speed:  INT;
	Fault:  BOOL;
END_VAR
VAR_OUTPUT
	Animation_B1:  BYTE;
	Color_B1:  BYTE;
	Speed_B1:  Byte;
	Animation_B2:  Byte;
	Color_B2:  Byte;
	Speed_B2:  BYTE;
END_VAR
VAR
END_VAR

//Commands for Light Bar

IF VTD_Mode = 0 AND NOT Fault THEN // (0)Disabled = No light  
    Animation_B1:= Animation_B2:= 0;
    
ELSIF VTD_Mode = 1 AND VTD_Speed = 0 AND  NOT Fault AND NOT "SinaSpeed_VTD_DB_1".EnableAxis THEN // (1)Manual= Yellow Stop
    Animation_B1 := Animation_B2 := 1;
    Color_B1 := Color_B2 := 4;
    
ELSIF VTD_Mode = 1 AND VTD_Speed > 0 AND VTD_Speed <= 33 AND  NOT Fault AND "SinaSpeed_VTD_DB_1".EnableAxis THEN // (1)Manual= Yellow until 33%
    Animation_B1 := Animation_B2 := 2;
    Speed_B1 := Speed_B2 := 2;
    Color_B1 := Color_B2 := 4;
    
ELSIF VTD_Mode = 1 AND VTD_Speed > 33 AND VTD_Speed <= 100 AND  NOT Fault THEN // (1)Manual= Yellow until 66%
    Animation_B1 := Animation_B2 := 2;
    Speed_B1 := Speed_B2 := 0;
    Color_B1 := Color_B2 := 4;
    
// ELSIF VTD_Mode = 1 AND VTD_Speed > 66 AND VTD_Speed <= 100 AND  NOT Fault THEN // (1)Manual= Yellow until 100%
//     Animation_B1 := Animation_B2 := 2;
//     Speed_B1 := Speed_B2 := 1;
//     Color_B1 := Color_B2 := 4;
    
ELSIF VTD_Mode = 2 AND VTD_Speed = 0 AND  NOT Fault AND NOT "SinaSpeed_VTD_DB_1".EnableAxis THEN // (2)Semi-auto = Blue Stop
    Animation_B1 := Animation_B2 := 1;
    Color_B1 := Color_B2 := 9;
    Speed_B1 := Speed_B2 := 0;
    
ELSIF VTD_Mode = 2 AND VTD_Speed > 0 AND VTD_Speed <= 33 AND  NOT Fault AND "SinaSpeed_VTD_DB_1".EnableAxis THEN // (2)Semi-auto = Blue until 33%
    Animation_B1 := Animation_B2 := 2;
    Speed_B1 := Speed_B2 := 2;
    Color_B1 := Color_B2 := 9;
    
ELSIF VTD_Mode = 2 AND VTD_Speed > 33 AND VTD_Speed <= 100 AND  NOT Fault THEN // (2)Semi-auto = Blue until 66%
    Animation_B1 := Animation_B2 := 2;
    Speed_B1 := Speed_B2 := 0;
    Color_B1 := Color_B2 := 9;
    
// ELSIF VTD_Mode = 2 AND VTD_Speed > 66 AND VTD_Speed <= 100 AND  NOT Fault THEN // (2)Semi-auto = Blue until 100%
//     Animation_B1 := Animation_B2 := 2;
//     Speed_B1 := Speed_B2 := 1;
//     Color_B1 := Color_B2 := 9;
    
ELSIF VTD_Mode = 3 AND VTD_Speed = 0 AND  NOT Fault AND NOT "SinaSpeed_VTD_DB_1".EnableAxis THEN // (3)Auto = Green Stop
    Animation_B1 := Animation_B2 := 1;
    Color_B1 := Color_B2 := 0;
    
ELSIF VTD_Mode = 3 AND VTD_Speed > 0 AND VTD_Speed <= 33 AND  NOT Fault AND "SinaSpeed_VTD_DB_1".EnableAxis THEN // (3)Auto = Green until 33%
    Animation_B1 := Animation_B2 := 2;
    Speed_B1 := Speed_B2 := 2;
    Color_B1 := Color_B2 := 0;
    
ELSIF VTD_Mode = 3 AND VTD_Speed > 33 AND VTD_Speed <= 100 AND  NOT Fault THEN // (3)Auto = Green until 66%
    Animation_B1 := Animation_B2 := 2;
    Speed_B1 := Speed_B2 := 0;
    Color_B1 := Color_B2 := 0;
    
// ELSIF VTD_Mode = 3 AND VTD_Speed > 66 AND VTD_Speed <= 100 AND  NOT Fault THEN // (3)Auto = Green until 100%
//     Animation_B1 := Animation_B2 := 2;
//     Speed_B1 := Speed_B2 := 1;
//     Color_B1 := Color_B2 := 0;
    
ELSIF VTD_Mode = 4 AND VTD_Speed = 0 AND  NOT Fault THEN // (4)Tech = Orange Stop
    Animation_B1 := Animation_B2 := 1;
    Color_B1 := Color_B2 := 2;
    
ELSIF VTD_Mode = 4 AND VTD_Speed > 0 AND VTD_Speed <= 33 AND  NOT Fault THEN // (4)Tech = Orange until 33%
    Animation_B1 := Animation_B2 := 2;
    Speed_B1 := Speed_B2 := 2;
    Color_B1 := Color_B2 := 2;
    
ELSIF VTD_Mode = 4 AND VTD_Speed > 33 AND VTD_Speed <= 66 AND  NOT Fault THEN // (4)Tech = Orange until 66%
    Animation_B1 := Animation_B2 := 2;
    Speed_B1 := Speed_B2 := 0;
    Color_B1 := Color_B2 := 2;
    
ELSIF VTD_Mode = 4 AND VTD_Speed > 66 AND VTD_Speed <= 100 AND  NOT Fault THEN // (4)Tech = Orange until 100%
    Animation_B1 := Animation_B2 := 2;
    Speed_B1 := Speed_B2 := 1;
    Color_B1 := Color_B2 := 2;
    
ELSIF VTD_Mode = 5 AND VTD_Speed = 0 AND  NOT Fault THEN // (5)Maintenance = White Stop
    Animation_B1 := Animation_B2 := 1;
    Color_B1 := Color_B2 := 19;
    
ELSIF VTD_Mode = 5 AND VTD_Speed > 0 AND VTD_Speed <= 33 AND  NOT Fault THEN // (5)Maintenance = White until 33%
    Animation_B1 := Animation_B2 := 2;
    Speed_B1 := Speed_B2 := 2;
    Color_B1 := Color_B2 := 19;
    
ELSIF VTD_Mode = 5 AND VTD_Speed > 33 AND VTD_Speed <= 66 AND  NOT Fault THEN // (5)Maintenance = White until 66%
    Animation_B1 := Animation_B2 := 2;
    Speed_B1 := Speed_B2 := 0;
    Color_B1 := Color_B2 := 19;
    
ELSIF VTD_Mode = 5 AND VTD_Speed > 66 AND VTD_Speed <= 100 AND  NOT Fault THEN // (5)Maintenance = White until 100%
    Animation_B1 := Animation_B2 := 2;
    Speed_B1 := Speed_B2 := 1;
    Color_B1 := Color_B2 := 19;
    
ELSIF Fault THEN // Fault = Flash Red
    Animation_B1:= Animation_B2 := 2;
    Color_B1:=Color_B2 := 1;
END_IF;

END_FUNCTION_BLOCK

// ---- POUs/VTD/VTD_FB.TcPOU
FUNCTION_BLOCK VTD_FB
VAR_INPUT
	System_no:  UINT;
	Safety_OK:  BOOL;
	Cnv_Sensors:  Cnv_Inputs_DUT;
	VTD_Settings:  VTD_Settings_DUT;
	Bypass_DP:  BOOL;
// 	Bypass:  Safety_Bypass_RemotePanel;
END_VAR
VAR_OUTPUT
END_VAR
VAR_IN_OUT
	VTD_Control:  VTD_Control_DUT;
	LE_Bypass_HMI:  BOOL;
END_VAR
VAR
	State:  UINT;
	Last_State:  UINT;
	I_State:  UInt;
	LD_Timer_1:  TON;
	LD_Timer:  TON;
	DP_Timer:  TON;
	Watchdog:  TON;
	CS_TImer:  TON;
	Interlock_Timer:  TON;
	MainSetpoint:  Int;
	Position_Offset:  Real;
	ChangeToLow:  Array[1..4] of DInt;
	DestPosition:  Real;
	SetUpSpeed:  UInt;
	LevelBelowExtractor:  UInt;
	IEC_Timer_0_Instance:  TON;
	DestinationLevel:  UInt;
	CurrentlLevel:  UInt;
	VTD_ID_Decoded:  ID_Decoded_DUT;
	Cnv_ID_Decoded:  ARRAY[1..2] OF ID_Decoded_DUT;
	IEC_Timer_0_Instance_1:  TON;
	IEC_Timer_0_Instance_2:  TON;
	VTD_ControlInstructionTask_ID_Old:  Int;
	R_Execulte:  R_TRIG;
	R_AutomatcMode:  R_TRIG;
	T_Encoders_Difference:  TON;
	T_LE_Error:  TON;
	T_Setpoint_Delay:  TON;
	Distance_mm:  Real;
	TravelTime_s:  UInt;
	LE_Prev_mm:  Real;
	DeltaPos_mm:  Real;
	SampleTime_s:  Real;
	VTDSpeed_mm_s:  Real;
	T_Speed:  TON;
	Speed_mm_per_percent:  Real;
	Speed_mm_s:  Real;
	TravelTime_ms:  UInt;
	Watchdog_PT:  Time;
	Position_OLD:  Real;
	R_Position_OLD:  R_TRIG;
END_VAR

VAR_TEMP
	Level_Accuracy:  STRING;
	i:  UINT;
	Upper_limit:  Bool;
	Ultimate_SlowDown:  Bool;
	Ultimate_Creep:  Bool;
	Lower_Limit:  Bool;
	Level_Detect:  Bool;
	Level_Detect1:  Bool;
	Level_Detect2:  Bool;
	DP2_Extended:  Bool;
	DP2_Retracted:  Bool;
	DP1_Extended:  Bool;
	DP1_Retracted:  Bool;
	Chain_Slack_1:  Bool;
	Chain_Slack_2:  Bool;
	Chain_Slack_3:  Bool;
	Chain_Slack_4:  Bool;
	DP1_Retract:  Bool;
	DP1_Extend:  Bool;
	DP2_Retract:  Bool;
	DP2_Extend:  Bool;
	Cnvs1_NotExtended:  Bool;
	Cnvs2_NotExtended:  Bool;
	Stoppers_NotExtended:  Bool;
	MainSetpoint1:  Int;
	HMI_Reset:  BOOL;
END_VAR

//Execute
R_Execulte(CLK := VTD_Control.Instruction.Execulte);

IF VTD_Control.Mode = 3 THEN
    VTD_Control.Instruction.Enable := TRUE;
END_IF;

VTD_Control.Enabled := VTD_Control.Instruction.Enable;

VTD_Control.Mode := VTD_Control.Instruction.Mode_Change;

IF NOT VTD_Control.Enabled AND NOT VTD_Control.Error THEN
    State := 0;
END_IF;

//MANUAL MODE
IF (VTD_Control.Mode = 1 OR VTD_Control.Mode = 5) AND NOT VTD_Control.Error AND VTD_Control.Enabled THEN
    State := 500;
END_IF;

(*
TODO:

Mode select is done via the HMI. Might add external mode select switches.
        
        Mode select mask:
        0: Disabled
        1: Manual
        2: Semi-Auto
        3: Auto
        4: Teach
        5: Maintenance
        
Device ID Format: XXYYZZ    
XX = Device type   
    01   VTD
    10  Cnv_Front_of_VTD
    11  Cnv_Rear_of_VTD
    12  Cnv_On_Extractor
    20  Safety_Stop_Front_of_VTD
    21  Safety_Stop_Rear_of_VTD
YY = Floor   
ZZ = VTD Connected to 
*)

{region "Sensor allocations"}
    //Assign inputs to local vars
    Upper_limit := VTD_Control.Inputs.Upper_limit;
    Ultimate_SlowDown := VTD_Control.Inputs.Ultimate_SlowDown;
    Ultimate_Creep := VTD_Control.Inputs.Ultimate_Creep;
    Lower_Limit := VTD_Control.Inputs.Lower_Limit;
    Level_Detect1 := VTD_Control.Inputs.Level_Detect1;
    Level_Detect2 := VTD_Control.Inputs.Level_Detect2;
    DP1_Extended := VTD_Control.Inputs.DP1_Extended;
    DP1_Retracted := VTD_Control.Inputs.DP1_Retracted;
    DP2_Extended := VTD_Control.Inputs.DP2_Extended;
    DP2_Retracted := VTD_Control.Inputs.DP2_Retracted;
    Chain_Slack_1 := VTD_Control.Inputs.Chain_Slack_1;
    Chain_Slack_2 := VTD_Control.Inputs.Chain_Slack_2;
    Chain_Slack_3 := VTD_Control.Inputs.Chain_Slack_3;
    Chain_Slack_4 := VTD_Control.Inputs.Chain_Slack_4;
    VTD_Control.LinearEnc := VTD_Control.Inputs.LE_Position;
    VTD_Control.AE := VTD_Control.Inputs.AE_Position_1;
{endregion}

{region "Cyclic Checks"}
    // Check for Pallet
    IF Cnv_Sensors.Forward_Sensor OR Cnv_Sensors.Backward_Sensor THEN
        VTD_Control.Pallet_Loaded := 1;//'Unknown';
    ELSE
        //No Pallet
        VTD_Control.Pallet_Loaded := 0;//'None';
    END_IF;
    
    //Docking pins
        IF DP1_Extended AND DP2_Extended THEN
            VTD_Control.LP_State := 1; //'Extended'
        ELSIF DP1_Retracted AND DP2_Retracted THEN
            VTD_Control.LP_State := 2; //'Retracted'
        ELSE
            VTD_Control.LP_State := 0; //'Unknown'
        END_IF;
        
        VTD_Control.DP_Extended := VTD_Control.LP_State = 1;
    
    // Level detect
    Level_Detect := Level_Detect1 AND Level_Detect2;
    
    //VTD extractor is docked
    IF DP1_Extended AND DP2_Extended AND Level_Detect AND
        (VTD_Control.LinearEnc - VTD_Settings.Teach_Values.Levels_LE[LevelBelowExtractor]) <= VTD_Settings.Level_Detect_LE THEN
        VTD_Control.Docked := TRUE;
    ELSE
        VTD_Control.Docked := FALSE;
    END_IF;
    
    //Ultimate stop checks
    IF (VTD_Control.LinearEnc < VTD_Settings.Slowdown_Count_LE OR VTD_Control.LinearEnc > VTD_Settings.Teach_Values.Levels_LE[VTD_Settings.Highest_Level] - VTD_Settings.Slowdown_Count_LE) AND
        Ultimate_Creep AND Ultimate_SlowDown AND VTD_Control.Running THEN
        VTD_Control.Motor_Speed := VTD_Settings.Creep_Speed;
        VTD_Control.Warning := 3; // Overtravel creep zone reached
    ELSIF (VTD_Control.LinearEnc < VTD_Settings.Slowdown_Count_LE OR VTD_Control.LinearEnc > VTD_Settings.Teach_Values.Levels_LE[VTD_Settings.Highest_Level] - VTD_Settings.Slowdown_Count_LE) AND
        NOT Ultimate_Creep AND Ultimate_SlowDown AND VTD_Control.Running THEN
        VTD_Control.Motor_Speed := VTD_Settings.Slow_Speed; // Overtravel slow zone reached
    END_IF;
    
    //Update Variables
    IF VTD_Control.Current_Task_Type = 0 OR VTD_Control.Current_Task_Type = 1 THEN
        VTD_Control.SM_State := State;
    ELSIF VTD_Control.Current_Task_Type = 2 OR VTD_Control.Current_Task_Type = 3 THEN
        VTD_Control.SM_State := I_State;
    END_IF;
    
    FOR i := VTD_Settings.Lowest_Level TO VTD_Settings.Highest_Level DO
        IF NOT Control.LCnv_Sys[System_no].Cnv_Level[i].Cnv1.Safety_Stop_Cnrl.Inputs.DP_Extended THEN
            Cnvs1_NotExtended := true;
        END_IF;
        IF NOT Control.LCnv_Sys[System_no].Cnv_Level[i].Cnv2.Safety_Stop_Cnrl.Inputs.DP_Extended THEN
            Cnvs2_NotExtended := true;
        END_IF;
    END_FOR;
    
    //Confirm whish level is below the extractor
    FOR i := VTD_Settings.Lowest_Level TO VTD_Settings.Highest_Level DO
        IF VTD_Control.LinearEnc >= (VTD_Settings.Teach_Values.Levels_LE[i] - VTD_Settings.Level_Detect_LE) THEN
            LevelBelowExtractor := i;
        END_IF;
    END_FOR;
    
    Stoppers_NotExtended := Cnvs1_NotExtended (*AND Cnvs2_NotExtended*);
    
    //AE ERROR
    IF VTD_Control.Inputs.AE_Status_2.15 THEN
        VTD_Control.AE_Error := 1;
    ELSE
        VTD_Control.AE_Error := 0;
    END_IF;
    
    //Encoder Delta
    VTD_Control.Encoder_Delta := ABS(VTD_Control.AE - VTD_Control.LinearEnc);
    
    //CURRENT LEVEL
    FOR i := VTD_Settings.Lowest_Level TO VTD_Settings.Highest_Level DO
        IF ABS(VTD_Control.LinearEnc - VTD_Settings.Teach_Values.Levels_LE[i]) <= VTD_Settings.VTD_Level_Granularity AND Level_Detect THEN
            VTD_Control.Current_Level := i;
            EXIT;
        ELSE
            VTD_Control.Current_Level := 0;
        END_IF;
    END_FOR;
    
    //SPEED mm/S
    T_Speed(IN := TRUE,
             PT := T#100MS);
    
    IF T_Speed.Q THEN
        DeltaPos_mm := ABS(VTD_Control.LinearEnc - LE_Prev_mm);
        VTDSpeed_mm_s := DeltaPos_mm / SampleTime_s;
        LE_Prev_mm := VTD_Control.LinearEnc;
        T_Speed(IN := FALSE,
                 PT := T#0MS);
    END_IF;
{endregion}

{region "Auto/Semi-Auto Mode"}
    CASE State OF
        0: //Idle
            Last_State := State;
            VTD_Control.Motor_UP := FALSE;
            VTD_Control.Motor_Down := FALSE;
            VTD_Control.Motor.Speed := 0;
            DestinationLevel := CurrentlLevel := 0;
            VTD_Control.Stopped := TRUE;
            Watchdog(IN := FALSE,
                          PT := T#0S);
            IF VTD_Control.Mode = 3 OR VTD_Control.Mode = 2 THEN
                IF VTD_Control.Instruction.Enable AND NOT VTD_Control.Error THEN
                    State := 10;
                END_IF;
            END_IF;
            
        10: //Standby
            Last_State := State;
            IF VTD_Control.Enabled AND NOT VTD_Control.Running AND VTD_Control.Instruction.Move_To_Level >= VTD_Settings.Lowest_Level AND
                VTD_Control.Instruction.Move_To_Level <= VTD_Settings.Highest_Level AND VTD_Control.Pallet_Loaded <> 1 AND
                ((VTD_Control.Instruction.Task_ID > 0 OR VTD_Control.Instruction.Task_Metadata <> '' AND VTD_Control.Mode = 3 AND Control.VTD_Order_Table[System_no].Task_Type = 1) OR
                (VTD_Control.Mode = 2 (*AND R_Execulte.Q*)))
            THEN
                IF VTD_Control.Instruction.Move_To_Level = VTD_Control.Current_Level AND VTD_Control.Instruction.Move_To_Level <> 0 THEN
                    VTD_Control.Warning := 1; //VTD already at level requested
                    VTD_Control.Instruction.Move_To_Level := 0;
                    //Go straght to the travel complete feedabck 
                ELSIF ((VTD_Control.Shuttle_Loaded = 0 OR VTD_Control.Shuttle_Loaded = 1) AND System_no <= 3)
                    OR System_no > 3
                THEN //EVERYTHING OK
                    DestinationLevel := VTD_Control.Instruction.Move_To_Level;
                    CurrentlLevel := VTD_Control.Current_Level;
                    VTD_Control.Current_Task_ID := VTD_Control.Instruction.Task_ID;
                    VTD_Control.Running := TRUE;
                    State := 20;
                END_IF;
            END_IF;

        20: //Extend all safety stoppers that are not in the up position
            Last_State := State;
            VTD_Control.Done := FALSE;// To report to order table
            FOR i := VTD_Settings.Lowest_Level TO VTD_Settings.Highest_Level DO
                IF NOT Control.LCnv_Sys[System_no].Cnv_Level[i].Cnv1.Safety_Stop_Cnrl.Inputs.DP_Extended THEN
                    Control.LCnv_Sys[System_no].Cnv_Level[i].Cnv1.Safety_Stop_Cnrl.Instruction.Extend := TRUE;
                END_IF;
                IF NOT Control.LCnv_Sys[System_no].Cnv_Level[i].Cnv2.Safety_Stop_Cnrl.Inputs.DP_Extended THEN
                    Control.LCnv_Sys[System_no].Cnv_Level[i].Cnv2.Safety_Stop_Cnrl.Instruction.Extend := TRUE;
                END_IF;
            END_FOR;
            State := 25;
            
        25: //Check to ensure the Safety stoppers are in the up position.
            Last_State := State;
            FOR i := VTD_Settings.Lowest_Level TO VTD_Settings.Highest_Level DO
                IF Control.LCnv_Sys[System_no].Cnv_Level[i].Cnv1.Safety_Stop_Cnrl.Inputs.DP_Extended THEN
                    Control.LCnv_Sys[System_no].Cnv_Level[i].Cnv1.Safety_Stop_Cnrl.Instruction.Extend := FALSE;
                END_IF;
                IF Control.LCnv_Sys[System_no].Cnv_Level[i].Cnv2.Safety_Stop_Cnrl.Inputs.DP_Extended THEN
                    Control.LCnv_Sys[System_no].Cnv_Level[i].Cnv2.Safety_Stop_Cnrl.Instruction.Extend := FALSE;
                END_IF;
            END_FOR;
            
            IF Control.LCnv_Sys[System_no].Cnv_Level[2].Cnv1.Safety_Stop_Cnrl.Inputs.DP_Extended AND
                Control.LCnv_Sys[System_no].Cnv_Level[3].Cnv1.Safety_Stop_Cnrl.Inputs.DP_Extended AND
                Control.LCnv_Sys[System_no].Cnv_Level[4].Cnv1.Safety_Stop_Cnrl.Inputs.DP_Extended AND
                Control.LCnv_Sys[System_no].Cnv_Level[5].Cnv1.Safety_Stop_Cnrl.Inputs.DP_Extended AND
                Control.LCnv_Sys[System_no].Cnv_Level[6].Cnv1.Safety_Stop_Cnrl.Inputs.DP_Extended AND
                Control.LCnv_Sys[System_no].Cnv_Level[2].Cnv2.Safety_Stop_Cnrl.Inputs.DP_Extended AND
                Control.LCnv_Sys[System_no].Cnv_Level[3].Cnv2.Safety_Stop_Cnrl.Inputs.DP_Extended AND
                Control.LCnv_Sys[System_no].Cnv_Level[4].Cnv2.Safety_Stop_Cnrl.Inputs.DP_Extended AND
                Control.LCnv_Sys[System_no].Cnv_Level[5].Cnv2.Safety_Stop_Cnrl.Inputs.DP_Extended AND
                Control.LCnv_Sys[System_no].Cnv_Level[6].Cnv2.Safety_Stop_Cnrl.Inputs.DP_Extended
            THEN
                State := 30;
            END_IF;
            
        30: //Undock the VTD
            Last_State := State;
            IF LevelBelowExtractor >= VTD_Settings.Lowest_Level AND LevelBelowExtractor < VTD_Settings.Highest_Level THEN
                IF VTD_Control.Docked OR
                    (VTD_Control.LinearEnc < VTD_Settings.Teach_Values.Levels_LE[LevelBelowExtractor] + 50) OR
                    (VTD_Control.LinearEnc < VTD_Settings.Teach_Values.Levels_LE[LevelBelowExtractor + 1] AND
                    VTD_Control.LinearEnc > VTD_Settings.Teach_Values.Levels_LE[LevelBelowExtractor + 1] - 10) THEN
                    IF VTD_Control.LP_State = 1 THEN //extended
                        VTD_Control.Motor_Speed := VTD_Settings.Dock_speed;
                        VTD_Control.Motor_UP := TRUE;
                        Position_Offset := VTD_Control.LinearEnc + 40;
                        State := 35;
                    ELSIF VTD_Control.LP_State = 2 THEN //retracted
                        State := 45;
                    ELSE //24:4 Docking pins in an known state
                        Set_Bit_F(Bit_Number := 5,
                                    Bit_Value := 1,
                                    Variavel := VTD_Control.VTD_Errors.Error_Word_2);
                    END_IF;
                ELSE
                    Position_Offset := VTD_Control.LinearEnc - 5;
                    State := 35;
                END_IF;
            ELSIF LevelBelowExtractor = VTD_Settings.Highest_Level THEN
                IF VTD_Control.Docked OR
                    (VTD_Control.LinearEnc < VTD_Settings.Teach_Values.Levels_LE[LevelBelowExtractor] + 50) THEN
                    IF VTD_Control.LP_State = 1 THEN //extended
                        VTD_Control.Motor_Speed := VTD_Settings.Dock_speed;
                        VTD_Control.Motor_UP := TRUE;
                        Position_Offset := VTD_Control.LinearEnc + 40;
                        State := 35;
                    ELSIF VTD_Control.LP_State = 2 THEN //retracted
                        State := 45;
                    ELSE //24:4 Docking pins in an known state
                        Set_Bit_F(Bit_Number := 5,
                                    Variavel := VTD_Control.VTD_Errors.Error_Word_2);
                    END_IF;
                ELSE
                    Position_Offset := VTD_Control.LinearEnc - 5;
                    State := 35;
                END_IF;
            END_IF;
            
        35: //Stop motor
            Last_State := State;
            IF NOT Level_Detect AND VTD_Control.LinearEnc >= Position_Offset THEN
                VTD_Control.Motor_Speed := 0;
                VTD_Control.Motor_UP := FALSE;
                State := 36;
            END_IF;
            
        36: //Retract the docking pins
            Last_State := State;
                DP2_Retract := DP1_Retract := TRUE;
                DP_Timer(IN := TRUE,
                          PT := UINT_TO_TIME(VTD_Settings.Lockpins_Timeout_Retract));
                
                IF DP2_Retracted THEN
                    DP2_Retract := FALSE;
                END_IF;
                IF VTD_Control.Inputs.DP1_Retracted THEN
                    DP1_Retract := FALSE;
                END_IF;
                
                IF VTD_Control.LP_State = 2 THEN
                    State := 40;
                END_IF;
                
            40: //Check docking pins have been retracted
                Last_State := State;
            IF VTD_Control.LP_State = 2 THEN
                DP_Timer(IN := FALSE,
                          PT := T#0S);
                DP2_Retract := DP1_Retract := FALSE;
                State := 45;
            END_IF;
            
        45: //Start moving towards the level required
            Last_State := State;
            //Check load type and set extractor speed
            IF VTD_Control.Shuttle_Loaded = 0 AND VTD_Control.Pallet_Loaded = 0 THEN
                VTD_Control.Motor_Speed := VTD_Settings.Empty_Speed;
            ELSIF VTD_Control.Shuttle_Loaded = 1 AND VTD_Control.Pallet_Loaded = 0 THEN
                VTD_Control.Motor_Speed := VTD_Settings.Shuttle_Speed;
            ELSIF VTD_Control.Shuttle_Loaded = 0 AND (VTD_Control.Pallet_Loaded > 0) THEN
                VTD_Control.Motor_Speed := VTD_Settings.Pallet_Speed;
            ELSIF VTD_Control.Shuttle_Loaded = 1 AND (VTD_Control.Pallet_Loaded > 0) THEN
                VTD_Control.Motor_Speed := VTD_Settings.Loaded_Speed;
            END_IF;
            
            DestPosition := VTD_Settings.Teach_Values.Levels_LE[VTD_Control.Instruction.Move_To_Level];
            SetUpSpeed := VTD_Control.Motor_Speed;
            
            // === DINAMIC WATCHDOG ===
            Speed_mm_s := SetUpSpeed * Speed_mm_per_percent;
            Distance_mm := ABS(DestPosition - VTD_Control.LinearEnc);
            
            //VTD needs to move up
            IF VTD_Control.LinearEnc < DestPosition THEN
                VTD_Control.Motor_UP := TRUE;
                State := 50;
                //VTD needs to move down
            ELSIF VTD_Control.LinearEnc > DestPosition THEN
                VTD_Control.Motor_Down := TRUE;
                State := 65; //change to 65
            END_IF;
            
        50: //travel upwards to designated level
            Last_State := State;
            ChangeToLow[1] := ABS((VTD_Settings.Slowdown_Count_LE / 100) * 80); (* 80% *) //80  600mm
            ChangeToLow[2] := ABS((VTD_Settings.Slowdown_Count_LE / 100) * 60); (* 60% *) //60
            ChangeToLow[3] := ABS((VTD_Settings.Slowdown_Count_LE / 100) * 40); (* 40% *) //40
            ChangeToLow[4] := ABS((VTD_Settings.Slowdown_Count_LE / 100) * 20); (* 20% *) //20 60
            
            //switch to fast freq Low UP
            IF ABS(DestPosition - VTD_Control.LinearEnc) > VTD_Settings.Slowdown_Count_LE THEN
                VTD_Control.Motor_Speed := SetUpSpeed; //5
                //switch to low freq
            ELSIF ABS(DestPosition - VTD_Control.LinearEnc) <= VTD_Settings.Slowdown_Count_LE
                AND ABS(DestPosition - VTD_Control.LinearEnc) > ChangeToLow[1] THEN
                VTD_Control.Motor_Speed := VTD_Settings.Slow_Calib_Speed * 1.8; //5 * 1.8 = 9%
            ELSIF ABS(DestPosition - VTD_Control.LinearEnc) <= ChangeToLow[1]
                AND ABS(DestPosition - VTD_Control.LinearEnc) > ChangeToLow[2] THEN
                VTD_Control.Motor_Speed := VTD_Settings.Slow_Calib_Speed * 1.6; //5 * 1.6 = 8%
            ELSIF ABS(DestPosition - VTD_Control.LinearEnc) <= ChangeToLow[2]
                AND ABS(DestPosition - VTD_Control.LinearEnc) > ChangeToLow[3] THEN
                VTD_Control.Motor_Speed := VTD_Settings.Slow_Calib_Speed * 1.4; //5 * 1.4 = 7%
            ELSIF ABS(DestPosition - VTD_Control.LinearEnc) <= ChangeToLow[3]
                AND ABS(DestPosition - VTD_Control.LinearEnc) > ChangeToLow[4] THEN
                VTD_Control.Motor_Speed := VTD_Settings.Slow_Calib_Speed * 1.2; //5 * 1.2 = 6%
            ELSIF ABS(DestPosition - VTD_Control.LinearEnc) <= ChangeToLow[4] THEN
                VTD_Control.Motor_Speed := VTD_Settings.Slow_Calib_Speed; //5%
                State := 55;
            END_IF;
            
            // Timeout in ms
            IF Speed_mm_s > 0 THEN
                TravelTime_ms := REAL_TO_UINT((Distance_mm / Speed_mm_s) * 1500.0);  // 1.5x safety factor
                IF TravelTime_ms < 5000 THEN
                    TravelTime_ms := 5000; // mínimum 5s
                END_IF;
            ELSE
                TravelTime_ms := 30000; // fallback 30s 
            END_IF;
            
            Watchdog_PT := UINT_TO_TIME(TravelTime_ms);
            
            Watchdog.TON(IN := TRUE,
                          PT := Watchdog_PT);
            
            
        55: // Travel upwards using slow speed towards required floor
            Last_State := State;
            IF VTD_Control.LinearEnc > VTD_Settings.Teach_Values.Levels_LE[VTD_Control.Instruction.Move_To_Level] - VTD_Settings.Creep_Count_LE
            THEN
                VTD_Control.Motor_Speed := VTD_Settings.Creep_Speed; //3% - 60mm 
                State := 60;
            END_IF;
            
        60: // Travel past the level in order to extend the docking pins
            Last_State := State;
            IF VTD_Control.LinearEnc > VTD_Settings.Teach_Values.Levels_LE[VTD_Control.Instruction.Move_To_Level] + VTD_Settings.Creep_Count_LE
            THEN
                VTD_Control.Motor_Speed := 0;
                VTD_Control.Motor_UP := FALSE;
                VTD_Control.Motor_Down := FALSE;
                State := 80;
            END_IF;
            
        65: //travel Downwards to designated level   
            Last_State := State;
            ChangeToLow[1] := ABS((VTD_Settings.Slowdown_Count_LE / 100) * 80); (* 80% *) //80
            ChangeToLow[2] := ABS((VTD_Settings.Slowdown_Count_LE / 100) * 60); (* 60% *) //60
            ChangeToLow[3] := ABS((VTD_Settings.Slowdown_Count_LE / 100) * 40); (* 40% *) //40
            ChangeToLow[4] := ABS((VTD_Settings.Slowdown_Count_LE / 100) * 20); (* 20% *) //20
            //switch to fast freq Low UP
            IF ABS(DestPosition - VTD_Control.LinearEnc) > VTD_Settings.Slowdown_Count_LE THEN
                VTD_Control.Motor_Speed := SetUpSpeed;
                //switch to low freq
            ELSIF ABS(DestPosition - VTD_Control.LinearEnc) <= VTD_Settings.Slowdown_Count_LE
                AND ABS(DestPosition - VTD_Control.LinearEnc) > ChangeToLow[1] THEN
                VTD_Control.Motor_Speed := REAL_TO_UINT(VTD_Settings.Slow_Calib_Speed * 1.8);
            ELSIF ABS(DestPosition - VTD_Control.LinearEnc) <= ChangeToLow[1]
                AND ABS(DestPosition - VTD_Control.LinearEnc) > ChangeToLow[2] THEN
                VTD_Control.Motor_Speed := REAL_TO_UINT(VTD_Settings.Slow_Calib_Speed * 1.6);
            ELSIF ABS(DestPosition - VTD_Control.LinearEnc) <= ChangeToLow[2]
                AND ABS(DestPosition - VTD_Control.LinearEnc) > ChangeToLow[3] THEN
                VTD_Control.Motor_Speed := REAL_TO_UINT(VTD_Settings.Slow_Calib_Speed * 1.4);
            ELSIF ABS(DestPosition - VTD_Control.LinearEnc) <= ChangeToLow[3]
                AND ABS(DestPosition - VTD_Control.LinearEnc) > ChangeToLow[4] THEN
                VTD_Control.Motor_Speed := REAL_TO_UINT(VTD_Settings.Slow_Calib_Speed * 1.2);
            ELSIF ABS(DestPosition - VTD_Control.LinearEnc) <= ChangeToLow[4] THEN
                VTD_Control.Motor_Speed := VTD_Settings.Slow_Calib_Speed;
                State := 70;
            END_IF;
            
            // Timeout in ms
            IF Speed_mm_s > 0 THEN
                TravelTime_ms := REAL_TO_UINT((Distance_mm / Speed_mm_s) * 2000.0);  // 1.5x safety factor
                IF TravelTime_ms < 5000 THEN
                    TravelTime_ms := 5000; // mínimum 5s
                END_IF;
            ELSE
                TravelTime_ms := 30000; // fallback 30s 
            END_IF;
            
            Watchdog_PT := UINT_TO_TIME(TravelTime_ms);
            
            Watchdog(IN := TRUE,
                     PT := Watchdog_PT);
            
        70: // Travel downwards using slow speed towards required floor 
            Last_State := State;
            IF VTD_Control.LinearEnc < VTD_Settings.Teach_Values.Levels_LE[VTD_Control.Instruction.Move_To_Level] + VTD_Settings.Creep_Count_LE
            THEN
                VTD_Control.Motor_Speed := 0;
                VTD_Control.Motor_UP := FALSE;
                VTD_Control.Motor_Down := FALSE;
                State := 80;
            END_IF;
            
        80: //Extend Docking pins
            Last_State := State;
            IF VTD_Control.LP_State = 2 AND NOT Level_Detect THEN
                DP1_Extend := DP2_Extend := TRUE;
                DP_Timer(IN := TRUE,
                          PT := UINT_TO_TIME(VTD_Settings.Lockpins_Timeout_Extend));
            ELSIF VTD_Control.LP_State <> 1 AND NOT Level_Detect THEN
                DP1_Extend := DP2_Extend := TRUE;
            ELSIF VTD_Control.LP_State = 1 THEN
                State := 85;
            END_IF;
            
            
        85: // Wait for docking pins to extend
            Last_State := State;
            IF VTD_Control.LP_State = 1 AND NOT Level_Detect THEN
                DP_Timer(IN := FALSE,
                          PT := T#0S);
                DP1_Extend := DP2_Extend := FALSE;
                VTD_Control.Motor_Speed := VTD_Settings.Dock_speed;
                VTD_Control.Motor_Down := TRUE;
                State := 90;
            END_IF;
            
        90: // Dock the VTD
            Last_State := State;
            //Using the LE for comparation and Release tension in the VTD chain
            IF ABS(VTD_Control.LinearEnc - DestPosition) <= (VTD_Settings.Level_Detect_LE) AND NOT CS_TImer.Q THEN
                CS_TImer(IN := TRUE,
                          PT := UINT_TO_TIME(VTD_Settings.Chain_Slack_Timeout));
            END_IF;
            IF CS_TImer.Q THEN
                VTD_Control.Motor_Speed := 0;
                VTD_Control.Motor_Down := FALSE;
                CS_TImer(IN := FALSE,
                          PT := T#0S);
                State := 95;
            END_IF;
            
        95: // Dock the VTD
            Last_State := State;
            //Check the level detect sensors
            IF (Level_Detect1 AND NOT Level_Detect2) OR
                (NOT Level_Detect1 AND Level_Detect2) THEN
                LD_Timer(IN := TRUE,
                          PT := UINT_TO_TIME(VTD_Settings.Level_Detect_Timeout));
            ELSIF NOT Level_Detect1 AND NOT Level_Detect2 THEN
                LD_Timer_1(IN := TRUE,
                            PT := UINT_TO_TIME(VTD_Settings.Level_Detect_Timeout * 5));
            ELSE
                LD_Timer(IN := FALSE,
                          PT := T#0S);
                LD_Timer_1(IN := FALSE,
                            PT := T#0S);
            END_IF;
            
            IF Level_Detect THEN
                Watchdog(IN := FALSE,
                          PT := T#0S);
                State := 100;
            END_IF;
            
        100: //Wait for Movement completion ack  
            Last_State := State;
            //Reset timers
            VTD_Control.Instruction.Move_To_Level := 0;
            DP_Timer(IN := FALSE,
                      PT := T#0S);
            Watchdog(IN := FALSE,
                      PT := T#0S);
            LD_Timer(IN := FALSE,
                      PT := T#0S);
            CS_TImer(IN := FALSE,
                      PT := T#0S);
            LD_Timer_1(IN := FALSE,
                        PT := T#0S);
            
            VTD_Control.Motor_Speed := 0;
            VTD_Control.Current_Task_ID := 0;
            VTD_Control.Running := FALSE;
            State := 0;
            
        400: // Error state
            VTD_Control.Instruction.Move_To_Level := 0;
            VTD_Control.Done := FALSE;// To report to order table
            VTD_Control.Motor.Enable := FALSE;
            VTD_Control.Motor_UP := FALSE;
            VTD_Control.Motor_Down := FALSE;
            VTD_Control.Running := FALSE;
            VTD_Control.Stopped := TRUE;
            VTD_Control.Motor.Speed := 0;
            VTD_Control.Motor.Forward := FALSE;
            VTD_Control.Motor.Reverse := FALSE;
            DP1_Extend := DP2_Extend := FALSE;
            DP1_Retract := DP2_Retract := FALSE;
            FOR i := VTD_Settings.Lowest_Level TO VTD_Settings.Highest_Level DO
                Control.LCnv_Sys[System_no].Cnv_Level[i].Cnv1.Safety_Stop_Cnrl.Instruction.Extend := FALSE;
                Control.LCnv_Sys[System_no].Cnv_Level[i].Cnv2.Safety_Stop_Cnrl.Instruction.Extend := FALSE;
            END_FOR;
            //Reset timers
            DP_Timer(IN := FALSE,
                      PT := T#0S);
            Watchdog(IN := FALSE,
                      PT := T#0S);
            LD_Timer(IN := FALSE,
                      PT := T#0S);
            CS_TImer(IN := FALSE,
                      PT := T#0S);
            LD_Timer_1(IN := FALSE,
                        PT := T#0S);
            IF VTD_Control.Instruction.Reset OR Reset_All OR HMI_Reset THEN
                VTD_Control.Error := FALSE;
                VTD_Control.Warning := 0;
                VTD_Control.Stopped := FALSE;
                VTD_Control.Current_Task_Type := 0;
                VTD_Control.VTD_Errors.Error_Word_1 := 0;
                VTD_Control.VTD_Errors.Error_Word_2 := 0;
                VTD_Control.VTD_Errors.Error_Word_3 := 0;
                VTD_Control.VTD_Errors.Error_Word_4 := 0;
                VTD_Control.VTD_Errors.Error_Word_5 := 0;
                State := 0;
            END_IF;
            
        500: //MANUAL MODE
            IF VTD_Control.Error = 0 AND VTD_Control.Enabled THEN
                //VTD
                IF VTD_Control.Instruction.Manual_Up AND NOT Upper_limit THEN
                    VTD_Control.Motor_UP := TRUE;
                    VTD_Control.Stopped := FALSE;
                    VTD_Control.Running := TRUE;
                    IF NOT (Ultimate_SlowDown OR Ultimate_Creep) THEN
                        VTD_Control.Motor_Speed := VTD_Settings.Manual_Speed;
                    END_IF;
                ELSIF VTD_Control.Instruction.Manual_Down AND NOT Lower_Limit THEN
                    VTD_Control.Motor_Down := TRUE;
                    VTD_Control.Stopped := FALSE;
                    VTD_Control.Running := TRUE;
                    IF VTD_Control.LinearEnc <= VTD_Settings.Teach_Values.Levels_LE[LevelBelowExtractor] + 300 AND VTD_Control.LP_State = 1 THEN
                        VTD_Control.Motor_Speed := VTD_Settings.Creep_Speed;
                    ELSIF NOT (Ultimate_SlowDown OR Ultimate_Creep) THEN
                        VTD_Control.Motor_Speed := VTD_Settings.Manual_Speed;
                    END_IF;
                ELSE
                    VTD_Control.Motor_Speed := 0;
                    VTD_Control.Stopped := TRUE;
                    VTD_Control.Running := FALSE;
                    VTD_Control.Motor_Down := FALSE;
                    VTD_Control.Motor_UP := FALSE;
                END_IF;
                
                //DOCKING PINS 2 
                IF NOT VTD_Control.Running AND VTD_Control.Instruction.Manual_LP_Extend
                    AND NOT DP2_Extended THEN
                    DP2_Extend := TRUE;
                ELSIF NOT VTD_Control.Running AND VTD_Control.Instruction.Manual_LP_Retract
                    AND NOT DP2_Retracted THEN
                    DP2_Retract := TRUE;
                ELSE
                    DP2_Extend := FALSE;
                    DP2_Retract := FALSE;
                END_IF;
                
                //DOCKING PINS 1 
                IF NOT VTD_Control.Running AND VTD_Control.Instruction.Manual_LP_Extend
                    AND NOT DP1_Extended THEN
                    DP1_Extend := TRUE;
                ELSIF NOT VTD_Control.Running AND VTD_Control.Instruction.Manual_LP_Retract
                    AND NOT DP1_Retracted THEN
                    DP1_Retract := TRUE;
                ELSE
                    DP1_Extend := FALSE;
                    DP1_Retract := FALSE;
                END_IF;
                
                IF VTD_Control.Mode <> 1 AND VTD_Control.Mode <> 5 THEN
                    State := 0;
                END_IF;
                
                IF DP2_Extend OR DP1_Extend THEN
                    DP_Timer(IN := TRUE,
                              PT := UINT_TO_TIME(VTD_Settings.Lockpins_Timeout_Extend));
                ELSIF DP2_Retract OR DP1_Retract THEN
                    DP_Timer(IN := TRUE,
                              PT := UINT_TO_TIME(VTD_Settings.Lockpins_Timeout_Retract));
                ELSE
                    DP_Timer(IN := FALSE,
                              PT := T0S);
                END_IF;
            END_IF;
    END_CASE;
{endregion}

{region "Shuttle Interlock"}
    // VTD needs to be in Auto mode to perform a Shuttle interlock
    CASE I_State OF
        0:
            IF VTD_Control.Mode = 3 AND VTD_Control.Shuttle_Interlock.Interlock_Request AND VTD_Control.Shuttle_Interlock.Shuttle_Interlock_Task_ID > 0 THEN
                I_State := 10;
            END_IF;
            
        10: //Standby
            
            //Start by decoding all the IDs of the devices pertaining to the VTD in question on that level
            "ID_Decode_F"(ID := VTD_Settings.ID,
                          ID_Decoded := VTD_ID_Decoded);
            "ID_Decode_F"(ID := "Settings_DB".LCnv_Sys[System_no].Cnv_Level[VTD_Control.Current_Level].Cnv1.ID,
                          ID_Decoded := Cnv_ID_Decoded[1]);
            "ID_Decode_F"(ID := "Settings_DB".LCnv_Sys[System_no].Cnv_Level[VTD_Control.Current_Level].Cnv2.ID,
                          ID_Decoded := Cnv_ID_Decoded[2]);
            
            // Ensure the VTD is in a state that it can perform an interlock
            IF VTD_Control.Docked AND NOT VTD_Control.Running AND (VTD_Control.Shuttle_Loaded = 0 OR VTD_Control.Shuttle_Loaded = 1) AND VTD_Control.Error = 0 THEN
                // Check to make sure the VTD and Shuttle are not both loaded
                IF VTD_Control.Pallet_Loaded = 1 THEN
                    VTD_Control.Warning := 1; // Both the VTD and Shuttles are loaded, can't perform the interlock
                ELSE
                    //Check that shuttle is on the correct floor, that the start location given and the shuttle actual position matches and the destination is the correct extractor barcode
                    IF (*VTD_Control.Current_Level = "Shuttle_MQTT_DB".Shuttle_MQTT[VTD_Control.Shuttle_Interlock.Shuttle_ID].Message.Shuttle_Status.Floor
                            AND*)VTD_Control.Shuttle_Interlock.Shuttle_Start_Location = "Shuttle_MQTT_DB".Shuttle_MQTT[VTD_Control.Shuttle_Interlock.Shuttle_ID].Message.Shuttle_Status.Position_ID
                            (*AND "Shuttle_MQTT_DB".Shuttle_MQTT[VTD_Control.Shuttle_Interlock.Shuttle_ID].Message.Shuttle_Status.Destination_ID = "Settings_DB".ECnv_Settings.Barcode_ID*)THEN
                        
                        //Check in which Buffer conveyor the shuttle is located
                        IF "Settings_DB".LCnv_Sys[System_no].Cnv_Level[VTD_Control.Current_Level].Cnv1.Barcode_ID =
                            VTD_Control.Shuttle_Interlock.Shuttle_Start_Location THEN
                            VTD_Control.Running := TRUE;
                            I_State := 20;
                        ELSIF "Settings_DB".LCnv_Sys[System_no].Cnv_Level[VTD_Control.Current_Level].Cnv2.Barcode_ID =
                            VTD_Control.Shuttle_Interlock.Shuttle_Start_Location THEN
                            VTD_Control.Running := TRUE;
                            I_State := 25;
                        ELSIF "Settings_DB".ECnv_Sys[System_no].Barcode_ID =
                            VTD_Control.Shuttle_Interlock.Shuttle_Start_Location AND
                            Control_GVL.VTD_Order_Table[System_no].Destination_Location = "Settings_DB".LCnv_Sys[System_no].Cnv_Level[VTD_Control.Current_Level].Cnv1.Barcode_ID THEN
                            VTD_Control.Running := TRUE;
                            I_State := 20;
                        ELSIF "Settings_DB".ECnv_Sys[System_no].Barcode_ID =
                            VTD_Control.Shuttle_Interlock.Shuttle_Start_Location AND
                            Control_GVL.VTD_Order_Table[System_no].Destination_Location = "Settings_DB".LCnv_Sys[System_no].Cnv_Level[VTD_Control.Current_Level].Cnv2.Barcode_ID THEN
                            VTD_Control.Running := TRUE;
                            I_State := 25;
                        ELSE
                            VTD_Control.Warning := 2; // Shuttle interlock start location not buffer conveyor of VTD
                        END_IF;
                    ELSE
                        VTD_Control.Warning := 3; // Cant interlock as shuttle and VTD level mismatch
                    END_IF;
                END_IF;
            ELSE
                VTD_Control.Warning := 4; // VTD not ready for interlock 
            END_IF;
            
            
        20: //Drop safety stops
            IF Cnv_ID_Decoded[1].Level = VTD_Control.Current_Level THEN
                Control.LCnv_Sys[System_no].Cnv_Level[VTD_Control.Current_Level].Cnv1.Safety_Stop_Cnrl.Instruction.Retract := TRUE;
                I_State := 30;
            ELSE
                VTD_Control.Error := TRUE; //24:16 Cannot find the correct safety pins to drop.
                Set_Bit_F(Bit_Number := 1,
                            Bit_Value := 1,
                            Variavel := VTD_Control.VTD_Errors.Error_Word_3);
                // I_State := 400;
            END_IF;
            
        25: //Drop safety pins   
            IF Cnv_ID_Decoded[2].Level = VTD_Control.Current_Level THEN
                Control.LCnv_Sys[System_no].Cnv_Level[VTD_Control.Current_Level].Cnv2.Safety_Stop_Cnrl.Instruction.Retract := TRUE;
                I_State := 35;
            ELSE
                VTD_Control.Error := TRUE; //24:16 Cannot find the correct safety pins to drop.
                Set_Bit_F(Bit_Number := 1,
                            Bit_Value := 1,
                            Variavel := VTD_Control.VTD_Errors.Error_Word_3);
                // I_State := 400;
            END_IF;
            //////////////////////////////////////////////////////////////////////////////////////////////////////////////////////////////////////////////////////////////////    
        30: //Confirm safety stops are down at the correct location
            //Send ready to interlock
            IF Control.LCnv_Sys[System_no].Cnv_Level[VTD_Control.Current_Level].Cnv1.Safety_Stop_Cnrl.LP_State = 0 THEN //RETRACTED
                Control.LCnv_Sys[System_no].Cnv_Level[VTD_Control.Current_Level].Cnv1.Safety_Stop_Cnrl.Instruction.Retract := FALSE;
                VTD_Control.Shuttle_Interlock.Ready_To_Interlock := TRUE;
                I_State := 40;
            END_IF;
            
        35: //Confirm safety stops are down at the correct location
            //Send ready to interlock
            IF Control.LCnv_Sys[System_no].Cnv_Level[VTD_Control.Current_Level].Cnv2.Safety_Stop_Cnrl.LP_State = 0 THEN //RETRACTED
                Control.LCnv_Sys[System_no].Cnv_Level[VTD_Control.Current_Level].Cnv2.Safety_Stop_Cnrl.Instruction.Retract := FALSE;
                VTD_Control.Shuttle_Interlock.Ready_To_Interlock := TRUE;
                I_State := 45;
            END_IF;
            ////////////////////////////////////////////////////////////////////////////////////////////////////////////////////////////////////////////////////////////////////
        40: //Wait for shuttle to move in or out VTD
            IF Control_GVL.VTD_Order_Table[System_no].Destination_Location = "Settings_DB".ECnv_Sys[System_no].Barcode_ID THEN
                IF "Settings_DB".ECnv_Sys[System_no].Barcode_ID = "Shuttle_MQTT_DB".Shuttle_MQTT[VTD_Control.Shuttle_Interlock.Shuttle_ID].Message.Shuttle_Status.Position_ID
                    AND "Shuttle_MQTT_DB".Shuttle_MQTT[VTD_Control.Shuttle_Interlock.Shuttle_ID].Message.Shuttle_Status.Operational_State = 'IDLE' THEN
                    Control.LCnv_Sys[System_no].Cnv_Level[VTD_Control.Current_Level].Cnv1.Safety_Stop_Cnrl.Instruction.Extend := TRUE;
                    I_State := 50;
                END_IF;
            ELSIF Control.VTD_Order_Table[System_no].Destination_Location = "Settings_DB".LCnv_Sys[System_no].Cnv_Level[VTD_Control.Current_Level].Cnv1.Barcode_ID THEN
                IF "Settings_DB".LCnv_Sys[System_no].Cnv_Level[VTD_Control.Current_Level].Cnv1.Barcode_ID = "Shuttle_MQTT_DB".Shuttle_MQTT[VTD_Control.Shuttle_Interlock.Shuttle_ID].Message.Shuttle_Status.Position_ID
                    AND "Shuttle_MQTT_DB".Shuttle_MQTT[VTD_Control.Shuttle_Interlock.Shuttle_ID].Message.Shuttle_Status.Operational_State = 'IDLE' THEN
                    Control.LCnv_Sys[System_no].Cnv_Level[VTD_Control.Current_Level].Cnv1.Safety_Stop_Cnrl.Instruction.Extend := TRUE;
                    I_State := 50;
                END_IF;
            END_IF;
            
        45: //Wait for shuttle to move in or out VTD
            IF Control_GVL.VTD_Order_Table[System_no].Destination_Location = "Settings_DB".ECnv_Sys[System_no].Barcode_ID THEN
                IF "Settings_DB".ECnv_Sys[System_no].Barcode_ID = "Shuttle_MQTT_DB".Shuttle_MQTT[VTD_Control.Shuttle_Interlock.Shuttle_ID].Message.Shuttle_Status.Position_ID
                    AND "Shuttle_MQTT_DB".Shuttle_MQTT[VTD_Control.Shuttle_Interlock.Shuttle_ID].Message.Shuttle_Status.Operational_State = 'IDLE' THEN
                    Control.LCnv_Sys[System_no].Cnv_Level[VTD_Control.Current_Level].Cnv2.Safety_Stop_Cnrl.Instruction.Extend := TRUE;
                    I_State := 55;
                END_IF;
            ELSIF Control.VTD_Order_Table[System_no].Destination_Location = "Settings_DB".LCnv_Sys[System_no].Cnv_Level[VTD_Control.Current_Level].Cnv2.Barcode_ID THEN
                IF "Settings_DB".LCnv_Sys[System_no].Cnv_Level[VTD_Control.Current_Level].Cnv2.Barcode_ID = "Shuttle_MQTT_DB".Shuttle_MQTT[VTD_Control.Shuttle_Interlock.Shuttle_ID].Message.Shuttle_Status.Position_ID
                    AND "Shuttle_MQTT_DB".Shuttle_MQTT[VTD_Control.Shuttle_Interlock.Shuttle_ID].Message.Shuttle_Status.Operational_State = 'IDLE' THEN
                    Control.LCnv_Sys[System_no].Cnv_Level[VTD_Control.Current_Level].Cnv2.Safety_Stop_Cnrl.Instruction.Extend := TRUE;
                    I_State := 55;
                END_IF;
            END_IF;
            //////////////////////////////////////////////////////////////////////////////////////////////////////////////////////////////////////////////////////////////////////////  
        50: //Check own sensors for shuttle/pallet state
            IEC_Timer_0_Instance_1(IN := TRUE,
                                    PT := T5S);
            IF Control.LCnv_Sys[System_no].Cnv_Level[VTD_Control.Current_Level].Cnv1.Safety_Stop_Cnrl.LP_State = 1 //EXTENDED
                THEN
                Control.LCnv_Sys[System_no].Cnv_Level[VTD_Control.Current_Level].Cnv1.Safety_Stop_Cnrl.Instruction.Extend := FALSE;
                VTD_Control.Shuttle_Interlock.Interlock_Complete := TRUE;
                I_State := 60;
            ELSIF IEC_Timer_0_Instance_1.Q THEN
                VTD_Control.Error := TRUE; //24:17 Error occured during interlock final check
                Set_Bit_F(Bit_Number := 2,
                            Bit_Value := 1,
                            Variavel := VTD_Control.VTD_Errors.Error_Word_3);
                I_State := 400;
            END_IF;
            
        55: //Check own sensors for shuttle/pallet state
            IEC_Timer_0_Instance_1(IN := TRUE,
                                    PT := T5S);
            IF Control.LCnv_Sys[System_no].Cnv_Level[VTD_Control.Current_Level].Cnv2.Safety_Stop_Cnrl.LP_State = 1 //EXTENDED
                THEN
                Control.LCnv_Sys[System_no].Cnv_Level[VTD_Control.Current_Level].Cnv2.Safety_Stop_Cnrl.Instruction.Extend := FALSE;
                VTD_Control.Shuttle_Interlock.Interlock_Complete := TRUE;
                I_State := 60;
            ELSIF IEC_Timer_0_Instance_1.Q THEN
                VTD_Control.Error := TRUE; //24:17 Error occured during interlock final check
                Set_Bit_F(Bit_Number := 2,
                            Bit_Value := 1,
                            Variavel := VTD_Control.VTD_Errors.Error_Word_3);
                I_State := 400;
            END_IF;
            
        60://Clear Vars
            IEC_Timer_0_Instance_1(IN := FALSE,
                                    PT := T0s);
            IEC_Timer_0_Instance_2(IN := FALSE,
                                    PT := T0s);
            IF VTD_Control.Shuttle_Interlock.Interlock_Complete_Ack THEN
                VTD_Control.Shuttle_Interlock.Ready_To_Interlock := FALSE;
                VTD_Control.Shuttle_Interlock.Interlock_Complete := FALSE;
                VTD_Control.Running := FALSE;
                I_State := 0;
            END_IF;
            
        400://ERROR MODE
            IEC_Timer_0_Instance_1(IN := FALSE,
                                    PT := T#0S);
            IEC_Timer_0_Instance_2(IN := FALSE,
                                    PT := T#0S);
            Interlock_Timer(IN := FALSE,
                             PT := T#0S);
            VTD_Control.Running := FALSE;
            VTD_Control.Shuttle_Interlock.Interlock_Complete := FALSE;
            VTD_Control.Shuttle_Interlock.Ready_To_Interlock := FALSE;
            Control.LCnv_Sys[System_no].Cnv_Level[VTD_Control.Current_Level].Cnv1.Safety_Stop_Cnrl.Instruction.Extend := FALSE;
            Control.LCnv_Sys[System_no].Cnv_Level[VTD_Control.Current_Level].Cnv2.Safety_Stop_Cnrl.Instruction.Extend := FALSE;
            Control.LCnv_Sys[System_no].Cnv_Level[VTD_Control.Current_Level].Cnv1.Safety_Stop_Cnrl.Instruction.Retract := FALSE;
            Control.LCnv_Sys[System_no].Cnv_Level[VTD_Control.Current_Level].Cnv2.Safety_Stop_Cnrl.Instruction.Retract := FALSE;
            IF VTD_Control.Instruction.Reset THEN
                VTD_Control.VTD_Errors.Error_Word_3 := 0;
                I_State := 0;
            END_IF;
    END_CASE;
    Interlock_Timer(IN := I_State >= 40 AND I_State <= 50,
                     PT := UINT_TO_TIME("Settings_DB".System.Shuttle_Interlock_Timeout) * 1000);
    
{endregion}


// IF System_no <> 3 THEN
{region "Cyclic Error Checks"}
    IF NOT Safety_OK THEN //SAFETY
        Set_Bit_F(Bit_Number := 0,
                  Variavel := VTD_Control.VTD_Errors.Error_Word_1);
    END_IF;
    
    IF VTD_Control.Instruction.Stop THEN //HMI STOP
        Set_Bit_F(Bit_Number := 1,
                    Variavel := VTD_Control.VTD_Errors.Error_Word_1);
    END_IF;
    
    IF NOT VTD_Control.Inputs.Upper_Overtravel AND NOT Bypass.Upper_limit THEN //UPPER OVERTRAVEL
        Set_Bit_F(Bit_Number := 2,
                    Variavel := VTD_Control.VTD_Errors.Error_Word_1);
    END_IF;
    
    IF NOT VTD_Control.Inputs.Lower_Overtravel AND NOT Bypass.Lower_limit THEN //LOWER OVERTRAVEL
        Set_Bit_F(Bit_Number := 3,
                    Variavel := VTD_Control.VTD_Errors.Error_Word_1);
    END_IF;
    
    //CHAIN SLACK
    IF Chain_Slack_1 AND NOT Bypass.Chain_Slack_1 THEN
        Set_Bit_F(Bit_Number := 0,
                    Variavel := VTD_Control.VTD_Errors.Error_Word_5);
    END_IF;
    
    IF Chain_Slack_2 AND NOT Bypass.Chain_Slack_2 THEN
        Set_Bit_F(Bit_Number := 1,
                    Variavel := VTD_Control.VTD_Errors.Error_Word_5);
    END_IF;
    
    IF Chain_Slack_3 AND NOT Bypass.Chain_Slack_3 THEN
        Set_Bit_F(Bit_Number := 2,
                    Variavel := VTD_Control.VTD_Errors.Error_Word_5);
    END_IF;
    
    IF Chain_Slack_4 AND NOT Bypass.Chain_Slack_4 THEN
        Set_Bit_F(Bit_Number := 3,
                    Variavel := VTD_Control.VTD_Errors.Error_Word_5);
    END_IF;
    
    //VFD ERROR
    IF VTD_Control.Motor.Error THEN
        Set_Bit_F(Bit_Number := 7,
                    Variavel := VTD_Control.VTD_Errors.Error_Word_4);
    END_IF;
    
    //HIGH LIMITS
    IF VTD_Control.LinearEnc > VTD_Settings.VTD_Max_Heigh AND NOT LE_Bypass_HMI AND NOT "VTD_HMI".LE_Bypass[System_no] THEN //21:5
        Set_Bit_F(Bit_Number := 4,
                    Variavel := VTD_Control.VTD_Errors.Error_Word_1);
    END_IF;
    
    IF VTD_Control.LinearEnc < VTD_Settings.VTD_Min_Height AND NOT LE_Bypass_HMI AND NOT "VTD_HMI".LE_Bypass[System_no] THEN //21:5
        Set_Bit_F(Bit_Number := 5,
                    Variavel := VTD_Control.VTD_Errors.Error_Word_1);
    END_IF;
    
    //AUTOMATIC MODE NOT DOCKED
    R_AutomatcMode(CLK := VTD_Control.Mode = 3);
    IF NOT VTD_Control.Docked AND R_AutomatcMode.Q THEN //22:1
        Set_Bit_F(Bit_Number := 8,
                    Variavel := VTD_Control.VTD_Errors.Error_Word_1);
    END_IF;
    
    IF NOT Level_Detect AND R_AutomatcMode.Q THEN //22:2
        Set_Bit_F(Bit_Number := 9,
                    Variavel := VTD_Control.VTD_Errors.Error_Word_1);
    END_IF;
    
    //TRYING RETRACT WHILE DOCKED
    IF VTD_Control.Docked AND (DP1_Retract OR DP2_Retract) THEN //22:5
        Set_Bit_F(Bit_Number := 12,
                    Variavel := VTD_Control.VTD_Errors.Error_Word_1);
    END_IF;
    
    //LE ERROR
    T_LE_Error.TON(IN := VTD_Control.Inputs.LE_Status.%X0 OR VTD_Control.Inputs.LE_Status.%X1 OR
                    VTD_Control.LinearEnc < VTD_Settings.VTD_Min_Height OR
                    VTD_Control.LinearEnc > VTD_Settings.VTD_Max_Heigh,
                    PT := t500ms);
    IF NOT LE_Bypass_HMI AND NOT "VTD_HMI".LE_Bypass[System_no] AND T_LE_Error.Q THEN
        Set_Bit_F(Bit_Number := 4,
                    Variavel := VTD_Control.VTD_Errors.Error_Word_3);
        T_LE_Error.TON(IN := FALSE,
                        PT := T0s);
    END_IF;
    
    
    
    //ABSOLUTE ENCODER
    IF VTD_Control.AE_Error > 0 THEN
        Set_Bit_F(Bit_Number := 5,
                    Variavel := VTD_Control.VTD_Errors.Error_Word_3);
        VTD_Control.Outputs.AE_Control_Word_1.7 := VTD_Control.Instruction.Reset OR Reset_All OR HMI_Reset;
    ELSE
        VTD_Control.Outputs.AE_Control_Word_1.7 := FALSE;
    END_IF;
    
    IEC_Timer_0_Instance(IN := VTD_Control.LinearEnc <= (VTD_Settings.Teach_Values.Levels_LE[LevelBelowExtractor] + 1) AND VTD_Control.Instruction.Manual_Down,
                          PT := T#300MS);
    
    //Errors while running
    IF VTD_Control.Running THEN
        IF LevelBelowExtractor < 7 THEN
            IF NOT (VTD_Control.LP_State = 2) AND // NOT 'Retracted'
                (VTD_Control.LinearEnc > (VTD_Settings.Teach_Values.Levels_LE[LevelBelowExtractor] + VTD_Settings.Slowdown_Count_LE) AND
                VTD_Control.LinearEnc < (VTD_Settings.Teach_Values.Levels_LE[LevelBelowExtractor + 1] - VTD_Settings.Creep_Count_LE) AND
                VTD_Control.Instruction.Manual_Up)
                OR
                IEC_Timer_0_Instance.Q
            THEN //22:4
                IF NOT Bypass_LP THEN
                    IF System_no <> 5 THEN
                        Set_Bit_F(Bit_Number := 11,
                                    Variavel := VTD_Control.VTD_Errors.Error_Word_1);
                    END_IF;
                END_IF;
            END_IF;
        ELSIF LevelBelowExtractor = 8 THEN
            IF NOT (VTD_Control.LP_State = 2) AND // NOT 'Retracted'
                (VTD_Control.LinearEnc > (VTD_Settings.Teach_Values.Levels_LE[LevelBelowExtractor] + VTD_Settings.Slowdown_Count_LE) AND
                VTD_Control.Instruction.Manual_Up)
                OR
                IEC_Timer_0_Instance.Q
            THEN //22:4
                IF NOT Bypass_LP THEN
                    IF System_no <> 5 THEN
                        Set_Bit_F(Bit_Number := 11,
                                    Variavel := VTD_Control.VTD_Errors.Error_Word_1);
                    END_IF;
                END_IF;
            END_IF;
        END_IF;
        
        IF VTD_Control.Motor.Error THEN //VFD ERROR
            Set_Bit_F(Bit_Number := 0,
                        Variavel := VTD_Control.VTD_Errors.Error_Word_4);
        ELSIF VTD_Control.LinearEnc_Error > 0 THEN //LE ERROR
            Set_Bit_F(Bit_Number := 1,
                        Variavel := VTD_Control.VTD_Errors.Error_Word_4);
        ELSIF VTD_Control.AE_Error > 0 THEN //AE ERROR
            Set_Bit_F(Bit_Number := 2,
                        Variavel := VTD_Control.VTD_Errors.Error_Word_4);
            
        ELSIF (DP1_Extended AND DP1_Retracted) OR (DP2_Extended AND DP2_Retracted) THEN // 25:4
            IF System_no <> 5 THEN
                Set_Bit_F(Bit_Number := 3,
                            Variavel := VTD_Control.VTD_Errors.Error_Word_4);
            ELSE
                ;
            END_IF;
        ELSIF Lower_Limit AND NOT Upper_limit AND NOT Bypass.Overtravel_Lower_limit THEN // 25:5
            Set_Bit_F(Bit_Number := 4,
                        Variavel := VTD_Control.VTD_Errors.Error_Word_4);
        ELSIF NOT Lower_Limit AND Upper_limit AND NOT Bypass.Overtravel_Upper_limit THEN // 25:6
            Set_Bit_F(Bit_Number := 5,
                        Variavel := VTD_Control.VTD_Errors.Error_Word_4);
        ELSIF Lower_Limit AND Upper_limit THEN // 25:7
            Set_Bit_F(Bit_Number := 6,
                        Variavel := VTD_Control.VTD_Errors.Error_Word_4);
        END_IF;
    END_IF;
    
    //Check if overtravel limit switches has been hit
    IF Upper_limit AND VTD_Control.Instruction.Manual_Up
    THEN //24:6 Top overtravel limit reached.
        Set_Bit_F(Bit_Number := 7,
                    Variavel := VTD_Control.VTD_Errors.Error_Word_2);
        IF VTD_Control.Mode = 2 OR VTD_Control.Mode = 3 THEN
            State := 400;
        ELSE
            State := 0;
        END_IF;
    ELSIF Lower_Limit AND VTD_Control.Instruction.Manual_Down
    THEN //24:7 Bottom overtravel limit reached.
        Set_Bit_F(Bit_Number := 8,
                    Variavel := VTD_Control.VTD_Errors.Error_Word_2);
        IF VTD_Control.Mode = 2 OR VTD_Control.Mode = 3 THEN
            State := 400;
        ELSE
            State := 0;
        END_IF;
    END_IF;
    
    //Need to monitor both encoders
    IF ABS(VTD_Control.Encoder_Delta) > VTD_Settings.Encoder_Delta_Warning THEN
        VTD_Control.Warning := 2;
    END_IF;
    
    T_Encoders_Difference(IN := ABS(VTD_Control.Encoder_Delta) > VTD_Settings.Encoder_Delta_Error,
                           PT := T#500MS);
    
    IF T_Encoders_Difference.Q AND NOT LE_Bypass_HMI AND NOT "VTD_HMI".LE_Bypass[System_no] THEN
        //Send error message that encoder error is to large
        Set_Bit_F(Bit_Number := 2,
                    Variavel := VTD_Control.VTD_Errors.Error_Word_2);
    END_IF;
    
    // Level detect timer 
    IF LD_Timer.Q OR LD_Timer_1.Q THEN
        LD_Timer(IN := FALSE,
                  PT := T#0S);
        LD_Timer_1(IN := FALSE,
                    PT := T#0S);
            Set_Bit_F(Bit_Number := 11,
                        Variavel := VTD_Control.VTD_Errors.Error_Word_4);
    END_IF;
    
    //Locking pin timer
    IF DP_Timer.Q AND (DP1_Retract OR DP1_Extend) THEN //24:2 Locking pins took to long to extend
        Set_Bit_F(Bit_Number := 3,
                    Variavel := VTD_Control.VTD_Errors.Error_Word_2);
    ELSIF DP_Timer.Q AND (DP2_Retract AND DP2_Extend) THEN //24:3 Locking pins took to long to retract
        Set_Bit_F(Bit_Number := 4,
                    Variavel := VTD_Control.VTD_Errors.Error_Word_2);
    END_IF;
    
    IF Interlock_Timer.Q THEN //Interlock process timed out
        Set_Bit_F(Bit_Number := 3,
                    Variavel := VTD_Control.VTD_Errors.Error_Word_3);
        I_State := 400;
    END_IF;
    
    //MOVIVENT VTD UNEXPECTED
    //Take the position old
    R_Position_OLD(CLK:= NOT VTD_Control.Motor_UP AND NOT VTD_Control.Motor_Down AND MainSetpoint1 = 0);
    
    IF R_Position_OLD.Q THEN
        Position_OLD := VTD_Control.LinearEnc;
    ELSIF NOT R_Position_OLD.CLK THEN
        Position_OLD := 0;
    END_IF;
    
    //VTD STILL MOVING
    IF ABS(VTD_Control.LinearEnc - Position_OLD) > Tol_VTD_Still_Moving THEN
        Set_Bit_F(Bit_Number := 6,
                    Variavel := VTD_Control.VTD_Errors.Error_Word_3);
    END_IF;
    
    // Watchdog bit
    // IF Watchdog.Q THEN
    //     VTD_Control.Running := FALSE;
    //     IF VTD_Control.Mode = 4 THEN //24:9 Teach timed out
    //         Set_Bit_F(Bit_Number := 10,
    //                     Bit_Value := 1,
    //                     Variavel := VTD_Control.VTD_Errors.Error_Word_2);
    //     ELSIF VTD_Control.Mode = 3 THEN //24:9 Auto timed out
    //         Set_Bit_F(Bit_Number := 10,
    //                     Bit_Value := 1,
    //                     Variavel := VTD_Control.VTD_Errors.Error_Word_2);
    //     ELSIF VTD_Control.Mode = 2 THEN //24:9 Semi auto timed out
    //         Set_Bit_F(Bit_Number := 10,
    //                     Bit_Value := 1,
    //                     Variavel := VTD_Control.VTD_Errors.Error_Word_2);
    //     END_IF;
    // END_IF;
    
    IF ((System_no = 1 AND "Errors_Profinet_1".%X8) OR
        (System_no = 2 AND "Errors_Profinet_3".%X7) OR
        (System_no = 3 AND "Errors_Profinet_5".%X4) OR
        (System_no = 4 AND "Errors_Profinet_7".%X1) OR
        (System_no = 5 AND "Errors_Profinet_8".%X6)) AND VTD_Control.Mode = 3
    THEN //Interface Profinet error
        Set_Bit_F(Bit_Number := 3,
                    Variavel := VTD_Control.VTD_Errors.Error_Word_3);
    END_IF;
    
    // go to error state
    IF VTD_Control.VTD_Errors.Error_Word_1 <> 0 OR
        VTD_Control.VTD_Errors.Error_Word_2 <> 0 OR
        VTD_Control.VTD_Errors.Error_Word_3 <> 0 OR
        VTD_Control.VTD_Errors.Error_Word_4 <> 0 OR
        VTD_Control.VTD_Errors.Error_Word_5 <> 0 THEN
        VTD_Control.Error := TRUE;
        State := 400;
    END_IF;
{endregion}
// END_IF;

